Yaskawa INFORM job: SKRZYNIA_5040_180_STOPNI_10B_NEW.JBI

/JOB
//NAME SKRZYNIA_5040_180_STOPNI_10B_NEW
///FOLDERNAME 02-SKRZYNIE_JOBS
//POS
///NPOS 627,627,0,26,0,0
///TOOL 0
///POSTYPE PULSE
///PULSE
C00000=-21231,-51303,42314,2367,6591,-1439
C00001=-12854,-61498,-6635,149088,-29435,16513
C00002=84284,-61498,-6635,149088,14842,16513
C00003=84426,-61498,-62039,149088,14842,16513
C00004=84426,-61498,-83719,149088,14842,16513
C00005=40079,-25830,-61904,72398,37828,17494
C00006=40079,-25830,-61904,72398,37828,17494
C00007=38824,-23395,-60038,72349,38727,17731
C00008=41545,-22667,-59464,70826,37145,18191
C00009=40079,-25830,-61904,72398,37828,17494
C00010=40079,-23879,-31232,97616,36989,2612
C00011=40241,-22903,-30855,97033,36795,2952
C00012=39596,-21803,-29985,96678,37187,3182
C00013=41542,-21522,-29763,96797,35874,3054
C00014=40241,-22903,-30855,97033,36795,2952
C00015=44500,-22967,-34027,49689,40772,15208
C00016=44759,-21950,-33222,49364,40770,15399
C00017=43898,-20603,-32137,49608,41392,15289
C00018=45676,-20288,-31878,48567,40497,15854
C00019=44759,-21950,-33222,49364,40770,15399
C00020=50639,-31838,-53853,40430,42590,20636
C00021=47737,-42531,-47731,84740,46626,-3202
C00022=73324,-51450,-15857,136644,48513,-27329
C00023=28578,-31257,-33285,101874,54895,-3139
C00024=29101,-23166,-41439,93785,52323,3372
C00025=30342,-16402,-40775,90158,51109,6027
C00026=29555,-14242,-38855,90054,51607,6222
C00027=31304,-14182,-38798,89754,50458,6198
C00028=30342,-16402,-40775,90158,51109,6027
C00029=37840,-26567,-47806,97824,39338,5403
C00030=38314,-22656,-45541,96192,38787,6352
C00031=38740,-21749,-44817,95954,38481,6451
C00032=38106,-20505,-43805,95701,38856,6673
C00033=39920,-20274,-43616,95549,37666,6573
C00034=38740,-21749,-44817,95954,38481,6451
C00035=35154,-23288,-28184,89821,43405,2441
C00036=35403,-21021,-26397,89340,43215,2751
C00037=34678,-19569,-25213,89063,43699,2948
C00038=36545,-19419,-25091,89018,42427,2940
C00039=35403,-21021,-26397,89340,43215,2751
C00040=46673,-28267,-59493,36306,49500,22578
C00041=47298,-25083,-54483,36432,48421,22382
C00042=46134,-23276,-53085,36983,49197,22170
C00043=48093,-22778,-52692,35651,48513,22818
C00044=47298,-25083,-54483,36432,48421,22382
C00045=43000,-32780,-49011,53703,41088,15214
C00046=66148,-65994,-55487,105361,28212,-7739
C00047=66148,-65994,-55487,105361,28212,-7739
C00048=59848,-54778,-49507,133915,29212,-10807
C00049=45497,-38347,-41839,114412,32622,-465
C00050=46376,-32635,-46933,102993,29107,5780
C00051=46303,-28031,-46898,97061,28371,8976
C00052=45038,-26161,-45521,96183,29128,9541
C00053=46946,-25787,-45238,96120,27855,9431
C00054=46303,-28031,-46898,97061,28371,8976
C00055=45864,-17128,1685,129467,40696,-9274
C00056=46023,-15894,1830,128891,40053,-8896
C00057=45181,-14790,2774,128176,40341,-8535
C00058=46921,-14545,2986,129317,39465,-9073
C00059=45402,-17127,796,128656,40504,-8810
C00060=42828,-21985,-11573,106778,34538,-1929
C00061=43349,-21404,-11124,106831,34165,-1930
C00062=42250,-19876,-9917,105946,34757,-1485
C00063=44494,-19460,-9583,106781,33302,-1837
C00064=42797,-21858,-11474,106726,34550,-1903
C00065=42956,-14057,7354,88292,32197,-569
C00066=43438,-13569,7781,88275,31880,-510
C00067=42549,-12302,8904,87823,32462,-349
C00068=44721,-11883,9282,88161,31033,-316
C00069=42944,-14884,6642,88491,32210,-682
C00070=72417,-64226,-72669,53660,37323,27470
C00071=81480,-74508,-67932,111005,17511,3722
C00072=42492,-36415,-29790,92406,42740,11684
C00073=29699,-14901,-14062,86637,51249,15251
C00074=28921,-12904,-12269,86425,51786,15406
C00075=30978,-12767,-12144,86426,50380,15429
C00076=29506,-17416,-16239,86937,51377,15018
C00077=88410,-69609,-60867,139529,19008,-8209
C00078=62412,-62489,-12046,-12266,17816,34850
C00079=0,-52280,40443,0,6876,0
C00080=-681,-52632,38645,-5695,5489,-631
C00081=-17840,-61498,-6635,-149088,-29435,-16513
C00082=-84284,-61498,-6635,-149088,14842,-16513
C00083=-84426,-61498,-62039,-149088,14842,-16513
C00084=-84426,-61498,-83719,-149088,14842,-16513
C00085=-83351,-27062,-60322,-167360,37385,6517
C00086=-83351,-27062,-60322,-167360,37385,23281
C00087=-45097,-23850,-79932,-76262,26943,-22849
C00088=-48253,-15729,-73342,-71138,25693,-24842
C00089=-50302,-13076,-73239,-65836,25323,-27140
C00090=-49401,-11675,-71961,-66260,25816,-27133
C00091=-50608,-11574,-71867,-65226,25249,-27391
C00092=-49660,-13361,-73494,-66442,25615,-26975
C00093=-48242,-21102,-77802,-73044,25430,-23851
C00094=-42432,-29691,-46140,-101591,34194,-3953
C00095=-40467,-32259,-45349,-89481,35752,-6083
C00096=-35590,-22323,-38089,-87474,43148,-7978
C00097=-34853,-20780,-36847,-87247,43643,-8181
C00098=-37029,-20471,-36594,-86926,42180,-8224
C00099=-35503,-23333,-38886,-87700,43207,-7835
C00100=-41659,-25848,-37197,-61468,39541,-12344
C00101=-42019,-23363,-32043,-63110,38591,-11327
C00102=-41283,-22167,-31102,-63128,39154,-11341
C00103=-43189,-21868,-30866,-62281,38009,-11788
C00104=-40846,-25460,-35158,-62968,39555,-11455
C00105=-39561,-32409,-42051,-71473,38885,-9254
C00106=-88477,-67032,-53890,-125185,13082,17955
C00107=-90715,-66667,-50935,-152816,24533,28486
C00108=-30735,-26920,-32844,-95116,50209,-1071
C00109=-37180,-24683,-31930,-114741,47007,2943
C00110=-36407,-19634,-34656,-109847,45004,-453
C00111=-38352,-16604,-33863,-108521,43129,-1176
C00112=-37479,-14809,-32279,-108169,43576,-1482
C00113=-39395,-14487,-31992,-108361,42368,-1194
C00114=-37253,-18321,-35339,-108644,43916,-1187
C00115=-30948,-19486,-27368,-89515,49970,-2899
C00116=-32453,-17458,-25663,-89179,48933,-3088
C00117=-31896,-16151,-24534,-89028,49305,-3221
C00118=-33527,-16125,-24510,-88960,48196,-3202
C00119=-31291,-18911,-26892,-89421,49733,-2955
C00120=-32789,-14788,-10714,-75998,48642,-1904
C00121=-33953,-13481,-9550,-75758,47902,-2112
C00122=-33380,-12226,-8408,-75670,48319,-2157
C00123=-35020,-12164,-8351,-75529,47228,-2306
C00124=-33300,-14767,-10697,-75957,48300,-1949
C00125=-33300,-14767,-10697,-75957,48300,-1949
C00126=-33901,-13199,-7224,-76945,47663,-1266
C00127=-33178,-11617,-5779,-76815,48184,-1329
C00128=-35129,-11426,-5603,-76688,46886,-1497
C00129=-32900,-14718,-9841,-76444,48459,-1584
C00130=-46324,-38325,-53351,-48650,39022,-16558
C00131=-84678,-53272,-42524,-56273,5220,-14251
C00132=-79949,-57830,-54545,-43165,18800,-25262
C00133=-85199,-63426,-59279,-35356,8253,-25340
C00134=-43240,-40066,-69296,-76804,34492,-13950
C00135=-32352,-24302,-62495,-76398,48702,-17646
C00136=-33867,-19497,-59989,-74208,48202,-18898
C00137=-33043,-17469,-58279,-74274,48770,-19034
C00138=-35172,-17180,-58031,-73305,47532,-19251
C00139=-33150,-20833,-61090,-74721,48572,-18687
C00140=-32525,-19963,-22291,-97454,48417,-2656
C00141=-34479,-17146,-19937,-97221,47013,-2812
C00142=-33716,-15515,-18525,-96928,47480,-3025
C00143=-35357,-15455,-18472,-97073,46375,-2908
C00144=-33341,-18474,-21063,-97306,47817,-2759
C00145=-32838,-10388,7981,-94473,48357,2926
C00146=-33747,-9461,8037,-94117,47673,2571
C00147=-33094,-8062,9377,-93861,48090,2458
C00148=-34952,-7927,9507,-94260,46861,2543
C00149=-33010,-10379,7174,-94037,48174,2591
C00150=-36099,-20774,-22249,-70758,44565,-7624
C00151=-37926,-16067,-12890,-73276,42575,-5996
C00152=-37323,-14944,-11908,-73188,43017,-6038
C00153=-39053,-14785,-11769,-72915,41882,-6255
C00154=-37847,-19214,-17221,-72670,42783,-6386
C00155=-73757,-59015,-49060,-81128,32509,-3444
C00156=-66351,-49775,-22313,-121187,42752,19491
C00157=-38126,-18978,-6321,-103556,42156,4232
C00158=-39485,-17529,-8330,-90200,39091,223
C00159=-38315,-15563,-6658,-89669,39866,-39
C00160=-40130,-15376,-6497,-89855,38637,-21
C00161=-40610,-23081,-12745,-91737,38407,1092
C00162=-82794,-45547,-18103,-153793,26453,27163
C00163=-46099,-67236,-11725,-98004,28606,19827
C00164=275,-40498,62911,330,272,-175
C00165=-21231,-51303,42314,2367,6591,-1439
C00166=-12854,-61498,-6635,149088,-29435,16513
C00167=84284,-61498,-6635,149088,14842,16513
C00168=84426,-61498,-62039,149088,14842,16513
C00169=84426,-61498,-83719,149088,14842,16513
C00170=40079,-25830,-61904,72398,37828,17494
C00171=43542,-21744,-53414,85694,32141,12908
C00172=43538,-20959,-59091,78847,32551,16732
C00173=40079,-23879,-31232,97616,36989,2612
C00174=41069,-22296,-36683,87871,35939,7163
C00175=41069,-20857,-27994,94343,36275,3375
C00176=40241,-22903,-30855,97033,36795,2952
C00177=44500,-22967,-34027,49689,40772,15208
C00178=37674,-14410,-29425,54908,51799,12689
C00179=37617,-13106,-20810,58248,49229,10178
C00180=44759,-21950,-33222,49364,40770,15399
C00181=50639,-31838,-53853,40430,42590,20636
C00182=47737,-42531,-47731,84740,46626,-3202
C00183=78713,-49095,-28754,133607,38203,-24422
C00184=28578,-31257,-33285,101874,54895,-3139
C00185=29101,-23166,-41439,93785,52323,3372
C00186=31163,-13872,-34138,92103,50752,4440
C00187=31163,-14064,-41434,88282,50498,7326
C00188=30342,-16402,-40775,90158,51109,6027
C00189=37840,-26567,-47806,97824,39338,5403
C00190=38314,-22656,-45541,96192,38787,6352
C00191=39658,-19881,-39017,99036,38353,4498
C00192=39658,-20227,-46296,93241,37598,7980
C00193=38740,-21749,-44817,95954,38481,6451
C00194=35154,-23288,-28184,89821,43405,2441
C00195=36302,-20456,-32356,81251,42995,6506
C00196=36302,-19046,-24537,85721,42698,3608
C00197=35403,-21021,-26397,89340,43215,2751
C00198=46673,-28267,-59493,36306,49500,22578
C00199=35383,-14910,-45807,52457,59655,19882
C00200=35383,-15025,-38926,54776,56903,17744
C00201=47298,-25083,-54483,36432,48421,22382
C00202=43000,-32780,-49011,53703,41088,15214
C00203=90538,-65158,-52413,145953,6697,-22013
C00204=90538,-65158,-52413,145953,6697,-22013
C00205=59848,-54778,-49507,133915,29212,-10807
C00206=45497,-38347,-41839,114412,32622,-465
C00207=46376,-32635,-46933,102993,29107,5780
C00208=38443,-20223,-37840,96971,39567,10287
C00209=38443,-20698,-44956,91660,38993,13539
C00210=46303,-28031,-46898,97061,28371,8976
C00211=45864,-17128,1685,129467,40696,-9274
C00212=38069,-7942,12691,120284,49952,-5070
C00213=38069,-11604,1369,116685,47266,-2469
C00214=45402,-17127,796,128656,40504,-8810
C00215=42828,-21985,-11573,106778,34538,-1929
C00216=33281,-15275,-13406,92642,47209,4970
C00217=33281,-12456,-2996,97026,47894,1870
C00218=42797,-21858,-11474,106726,34550,-1903
C00219=42956,-14057,7354,88292,32197,-569
C00220=35915,-8349,8335,81338,43542,2014
C00221=35915,-4149,20758,86814,43229,-1568
C00222=42944,-14884,6642,88491,32210,-682
C00223=72417,-64226,-72669,53660,37323,27470
C00224=81480,-74508,-67932,111005,17511,3722
C00225=31559,-23192,-27729,97069,50041,14774
C00226=34278,-17590,-29530,108925,47275,14558
C00227=34921,-13948,-26935,108215,46513,15013
C00228=34921,-14719,-34056,104413,45059,17611
C00229=33936,-16225,-25259,110400,48238,13526
C00230=30729,-14807,-22031,91030,50318,16982
C00231=30729,-13019,-13516,94566,50766,14318
C00232=88410,-69609,-60867,139529,19008,-8209
C00233=62412,-62489,-12046,-12266,17816,34850
C00234=0,-52280,40443,0,6876,0
C00235=-681,-52632,38645,-5695,5489,-631
C00236=-17840,-61498,-6635,-149088,-29435,-16513
C00237=-84284,-61498,-6635,-149088,14842,-16513
C00238=-84426,-61498,-62039,-149088,14842,-16513
C00239=-84426,-61498,-83719,-149088,14842,-16513
C00240=-83351,-27062,-60322,-167360,37385,6517
C00241=-83351,-27062,-60322,-167360,37385,23281
C00242=-45097,-23850,-79932,-76262,26943,-22849
C00243=-48253,-15729,-73342,-71138,25693,-24842
C00244=-42869,-6204,-67496,-75794,33821,-25861
C00245=-42869,-3205,-70686,-69723,34977,-29338
C00246=-49660,-13361,-73494,-66442,25615,-26975
C00247=-48242,-21102,-77802,-73044,25430,-23851
C00248=-42432,-29691,-46140,-101591,34194,-3953
C00249=-40467,-32259,-45349,-89481,35752,-6083
C00250=-32032,-15700,-34761,-86363,49905,-9645
C00251=-32032,-14866,-27372,-89947,49973,-6979
C00252=-35503,-23333,-38886,-87700,43207,-7835
C00253=-41659,-25848,-37197,-61468,39541,-12344
C00254=-32550,-13183,-23016,-68651,53358,-8526
C00255=-34023,-12481,-22084,-63241,53452,-9524
C00256=-40846,-25460,-35158,-62968,39555,-11455
C00257=-39561,-32409,-42051,-71473,38885,-9254
C00258=-88477,-67032,-53890,-125185,13082,17955
C00259=-90715,-66667,-50935,-152816,24533,28486
C00260=-30735,-26920,-32844,-95116,50209,-1071
C00261=-37180,-24683,-31930,-114741,47007,2943
C00262=-36407,-19634,-34656,-109847,45004,-453
C00263=-39264,-14095,-28560,-110319,43249,69
C00264=-39254,-14742,-35710,-105973,41627,-2729
C00265=-37253,-18321,-35339,-108644,43916,-1187
C00266=-30948,-19486,-27368,-89515,49970,-2899
C00267=-33188,-17217,-33290,-80523,49125,-7157
C00268=-33231,-16133,-25752,-84153,48705,-4513
C00269=-31291,-18911,-26892,-89421,49733,-2955
C00270=-32789,-14788,-10714,-75998,48642,-1904
C00271=-32456,-10000,-8763,-74569,51725,-2878
C00272=-32456,-7502,814,-78111,50801,-165
C00273=-33300,-14767,-10697,-75957,48300,-1949
C00274=-33300,-14767,-10697,-75957,48300,-1949
C00275=-31039,-7597,-4415,-75714,54029,-1891
C00276=-31745,-5891,1281,-74609,53027,-1007
C00277=-32900,-14718,-9841,-76444,48459,-1584
C00278=-46324,-38325,-53351,-48650,39022,-16558
C00279=-84678,-53272,-42524,-56273,5220,-14251
C00280=-79949,-57830,-54545,-43165,18800,-25262
C00281=-85199,-63426,-59279,-35356,8253,-25340
C00282=-43240,-40066,-69296,-76804,34492,-13950
C00283=-32352,-24302,-62495,-76398,48702,-17646
C00284=-34311,-15084,-43386,-89458,46770,-12174
C00285=-34303,-14562,-49859,-85086,46777,-15220
C00286=-33150,-20833,-61090,-74721,48572,-18687
C00287=-32525,-19963,-22291,-97454,48417,-2656
C00288=-35706,-13608,-12356,-102024,46946,-662
C00289=-35706,-15621,-21438,-97808,45877,-3577
C00290=-33341,-18474,-21063,-97306,47817,-2759
C00291=-32838,-10388,7981,-94473,48357,2926
C00292=-33093,-7396,5806,-90907,49596,566
C00293=-33114,-3922,16616,-94789,50065,3444
C00294=-33010,-10379,7174,-94037,48174,2591
C00295=-36099,-20774,-22249,-70758,44565,-7624
C00296=-34715,-11750,-12273,-72011,49148,-6727
C00297=-34715,-9605,-3694,-75523,48112,-4187
C00298=-37847,-19214,-17221,-72670,42783,-6386
C00299=-73757,-59015,-49060,-81128,30370,-3444
C00300=-66351,-49775,-22313,-115582,40632,19491
C00301=-39230,-13378,9505,-118180,46878,7841
C00302=-45382,-7236,12023,-133378,48537,9962
C00303=-45404,-10871,608,-130166,44845,7725
C00304=-39289,-13633,5656,-114159,44810,6160
C00305=-38323,-13232,3563,-106275,42852,3854
C00306=-39624,-12309,2722,-105485,41613,3229
C00307=-39624,-8328,14658,-110578,43519,6514
C00308=-36264,-16485,7382,-110054,45980,6615
C00309=-44249,-32643,-4456,-118298,43922,12613
C00310=-31781,-48654,10305,-108801,40875,18482
C00311=275,-40498,62911,330,272,-175
C00312=-21231,-51303,42314,2367,6591,-1439
C00313=-12854,-61498,-6635,149088,-29435,16513
C00314=32880,-72586,-50560,79734,53940,25582
C00315=76664,-93599,-96338,114349,24908,7990
C00316=72545,-76403,-90681,98079,12187,16258
C00317=68435,-42241,-79282,43384,21203,43145
C00318=65057,-16377,-54230,51764,24572,24912
C00319=65057,-16377,-54230,51764,24572,24912
C00320=63338,-14509,-52578,53100,25585,24479
C00321=65493,-13068,-51269,50530,24633,25485
C00322=65057,-16377,-54230,51764,24572,24912
C00323=65057,-15356,-24189,99795,20011,765
C00324=64877,-14372,-23690,98704,20045,1316
C00325=64002,-13489,-22890,98156,20604,1621
C00326=65592,-12702,-22173,98357,19527,1466
C00327=64877,-14372,-23690,98704,20045,1316
C00328=68341,-13254,-25781,29903,31229,25524
C00329=68283,-12212,-24821,29865,31356,25548
C00330=67188,-11145,-23825,30867,31841,25051
C00331=68624,-10377,-23095,29361,31405,25809
C00332=68283,-12212,-24821,29865,31356,25548
C00333=67373,-28813,-51747,26561,36937,27500
C00334=65665,-56911,-59086,75825,31170,1181
C00335=86238,-56758,-47218,93606,16664,-7096
C00336=86238,-56758,-47218,93606,16664,-7096
C00337=58162,-25487,-29222,106212,35121,-6052
C00338=54729,-17550,-36821,90686,35172,3055
C00339=53879,-10723,-35593,84994,35691,6442
C00340=52628,-8898,-33837,85063,36512,6546
C00341=54193,-8333,-33282,84633,35489,6620
C00342=53879,-10723,-35593,84994,35691,6442
C00343=63265,-18185,-41125,95483,22448,4389
C00344=62561,-14368,-38517,92984,22773,5727
C00345=62689,-13396,-37636,92694,22678,5861
C00346=61812,-12400,-36718,92465,23238,6064
C00347=63331,-11679,-36046,92201,22238,6052
C00348=62689,-13396,-37636,92694,22678,5861
C00349=60836,-16142,-22303,87853,25853,3109
C00350=60346,-13901,-20318,87240,26185,3441
C00351=59279,-12702,-19226,86999,26911,3593
C00352=60868,-12050,-18626,86765,25831,3679
C00353=60346,-13901,-20318,87240,26185,3441
C00354=71174,-16943,-50501,16787,44328,31924
C00355=70846,-13961,-45205,17496,43056,31510
C00356=69412,-12602,-43961,18675,43507,30969
C00357=70949,-11616,-43043,17320,43301,31610
C00358=70846,-13961,-45205,17496,43056,31510
C00359=66765,-25643,-43957,33958,30926,25005
C00360=89904,-51519,-74342,14421,36812,44678
C00361=59533,-60921,-66479,83565,41795,11392
C00362=74572,-27669,-34920,136415,14797,-11887
C00363=72479,-21736,-38943,108586,11547,1590
C00364=70901,-17325,-38411,94105,11830,8638
C00365=69318,-15905,-37172,92885,12849,9347
C00366=70820,-15051,-36412,92531,11846,9399
C00367=70901,-17325,-38411,94105,11830,8638
C00368=70927,-7523,10343,151197,29871,-19432
C00369=70517,-6236,10737,150221,29352,-18933
C00370=69462,-5331,11645,148944,29606,-18324
C00371=70849,-4645,12343,150548,29173,-19084
C00372=70402,-7634,9356,150158,29478,-18907
C00373=68660,-13051,-4106,122816,18275,-8999
C00374=68895,-12351,-3471,122899,18094,-9031
C00375=67458,-11121,-2337,120787,18802,-8043
C00376=69212,-10147,-1425,122703,17774,-8922
C00377=68590,-12934,-4000,122687,18305,-8939
C00378=67960,-5141,15741,92957,15720,-628
C00379=68207,-4523,16370,92944,15555,-601
C00380=67051,-3465,17460,92338,16311,-404
C00381=68762,-2475,18496,92897,15183,-531
C00382=68227,-5981,14898,93242,15553,-745
C00383=75423,-38775,-29488,68062,11357,11878
C00384=83800,-53438,-37305,103753,25026,-1265
C00385=73693,-43023,-29306,101200,31062,8332
C00386=57182,-8361,13896,122065,42938,1264
C00387=54175,-4244,10116,111777,38351,4895
C00388=53015,-2664,11762,111180,39035,5172
C00389=54334,-2350,12093,111780,38228,4906
C00390=54175,-4244,10116,111777,38351,4895
C00391=89016,-59505,-36896,143842,20811,-11822
C00392=0,-52280,40443,0,6876,0
C00393=-681,-52632,38645,-5695,5489,-631
C00394=-17840,-61498,-6635,-149088,-29435,-16513
C00395=-84284,-61498,-6635,-149088,14842,-16513
C00396=-57949,-92832,-68327,-119114,39180,-13331
C00397=-51160,-78996,-68705,-103851,38676,-21739
C00398=-70129,-12201,-70194,-45988,15849,-32683
C00399=-70861,-4247,-62448,-43170,16032,-33903
C00400=-72229,-1292,-61598,-37253,16795,-36501
C00401=-71164,-286,-60510,-39045,17142,-35862
C00402=-72168,114,-60071,-37345,16819,-36474
C00403=-71747,-1710,-62044,-38091,16943,-36199
C00404=-72086,-8949,-67137,-41785,15362,-34318
C00405=-68226,-19972,-38714,-103620,16923,-1218
C00406=-67549,-22986,-38612,-80975,17520,-9124
C00407=-60286,-14955,-31870,-81576,26630,-9634
C00408=-59206,-13694,-30736,-81541,27366,-9725
C00409=-61026,-12796,-29913,-80837,26167,-9971
C00410=-60502,-15936,-32740,-81790,26471,-9505
C00411=-66711,-16726,-29834,-42060,26790,-21996
C00412=-66477,-14329,-24475,-44917,25565,-20507
C00413=-65503,-13376,-23611,-45716,26132,-20127
C00414=-67048,-12587,-22889,-44009,25442,-20959
C00415=-66009,-16611,-27996,-44380,26285,-20808
C00416=-67084,-23473,-35621,-52822,22843,-18344
C00417=-54372,-63877,-56403,-90862,27079,1323
C00418=-55608,-75012,-34654,-126966,55573,20814
C00419=-55608,-75012,-34654,-126966,55573,20814
C00420=-58069,-20780,-28125,-95622,31565,-134
C00421=-62818,-16895,-25617,-123146,31403,8811
C00422=-60301,-12189,-28106,-114654,29999,4030
C00423=-61167,-8731,-26593,-112607,28768,2985
C00424=-59960,-7252,-25135,-111997,29446,2563
C00425=-61574,-6413,-24296,-112502,28453,2957
C00426=-60636,-10677,-28466,-112685,29164,2987
C00427=-55814,-13636,-22293,-87541,33030,-3263
C00428=-56566,-11270,-20110,-87077,32519,-3496
C00429=-55709,-10167,-19066,-86969,33101,-3589
C00430=-57154,-9687,-18605,-86794,32120,-3632
C00431=-55949,-12989,-21706,-87412,32939,-3330
C00432=-57109,-8613,-4995,-71756,32687,-5152
C00433=-57764,-7017,-3429,-71410,32292,-5358
C00434=-56909,-5946,-2356,-71529,32873,-5273
C00435=-58347,-5433,-1836,-71115,31941,-5534
C00436=-57555,-8453,-4841,-71622,32398,-5235
C00437=-57555,-8453,-4841,-71622,32398,-5235
C00438=-57844,-6749,-1100,-73475,31868,-4209
C00439=-56760,-5394,262,-73573,32605,-4123
C00440=-58439,-4668,1002,-73167,31507,-4396
C00441=-57269,-8513,-4090,-72514,32435,-4729
C00442=-74194,-26905,-45748,-21164,30431,-30370
C00443=-93036,-61583,-83098,-4972,39040,-38907
C00444=-93036,-61583,-83098,-4972,39040,-38907
C00445=-71878,-28414,-61729,-48672,19032,-25171
C00446=-58025,-17185,-56692,-61796,34178,-22014
C00447=-58138,-12270,-53641,-59720,34855,-23185
C00448=-56898,-10637,-52111,-60384,35596,-23031
C00449=-58712,-9745,-51261,-58987,34681,-23500
C00450=-57851,-13714,-54968,-60141,34926,-22995
C00451=-57767,-13689,-16896,-100181,31334,-836
C00452=-58645,-10437,-13885,-99794,30663,-1040
C00453=-57513,-9065,-12573,-99347,31388,-1300
C00454=-58947,-8556,-12078,-99591,30423,-1148
C00455=-58031,-12031,-15383,-99926,31110,-974
C00456=-57646,-4162,14084,-101426,32077,4804
C00457=-58050,-2999,14481,-100683,31666,4357
C00458=-57067,-1784,15765,-100255,32298,4198
C00459=-58672,-1130,16464,-100866,31256,4407
C00460=-57676,-4116,13320,-100600,31921,4338
C00461=-61201,-13510,-16039,-60848,29053,-13371
C00462=-61885,-8475,-5914,-65722,27292,-10768
C00463=-61040,-7537,-4993,-65975,27855,-10622
C00464=-62506,-6917,-4380,-65230,26947,-11038
C00465=-62587,-11561,-10517,-63923,27184,-11731
C00466=-69972,-70945,-58827,-87515,35615,-17
C00467=-69972,-70945,-58827,-87515,35615,-17
C00468=-64053,-11295,342,-114563,25508,8776
C00469=-64305,-9514,-1154,-92513,22236,350
C00470=-62690,-7882,422,-91839,23314,70
C00471=-64201,-7220,1072,-92034,22288,112
C00472=-67149,-14673,-5883,-94845,20391,1413
C00473=-66017,-67071,-29713,-134523,32873,22112
C00474=-46099,-67236,-11725,-98004,28606,19827
C00475=275,-40498,62911,330,272,-175
C00476=-21231,-51303,42314,2367,6591,-1439
C00477=-12854,-61498,-6635,149088,-29435,16513
C00478=84284,-61498,-6635,149088,14842,16513
C00479=84426,-61498,-62039,149088,14842,16513
C00480=84426,-61498,-83719,149088,14842,16513
C00481=65057,-16377,-54230,51764,24572,24912
C00482=84197,-12836,-45810,-45141,8815,68584
C00483=84197,-12041,-51210,-30828,12194,61758
C00484=65057,-15356,-24189,99795,20011,765
C00485=74080,-15423,-30907,69143,7686,14038
C00486=74080,-14352,-23480,100923,7503,-991
C00487=64877,-14372,-23690,98704,20045,1316
C00488=68341,-13254,-25781,29903,31229,25524
C00489=74439,-11496,-26749,13621,29642,33649
C00490=74439,-10401,-19085,15788,25340,32499
C00491=68283,-12212,-24821,29865,31356,25548
C00492=75452,-19560,-44582,17787,36745,31835
C00493=68183,-44834,-62310,40554,34116,19994
C00494=94103,-63119,-69903,16230,17694,31762
C00495=91219,-55958,-51219,93435,14423,-1742
C00496=58162,-25487,-29222,106212,35121,-6052
C00497=54729,-17550,-36821,90686,35172,3055
C00498=70769,-15160,-35297,83470,11760,4000
C00499=70769,-15377,-40609,67973,12489,11436
C00500=53879,-10723,-35593,84994,35691,6442
C00501=63265,-18185,-41125,95483,22448,4389
C00502=62561,-14368,-38517,92984,22773,5727
C00503=77715,-13962,-33882,144680,4496,-21400
C00504=77806,-14046,-41277,60589,2532,18064
C00505=62689,-13396,-37636,92694,22678,5861
C00506=60836,-16142,-22303,87853,25853,3109
C00507=74678,-16514,-29029,42946,9451,23276
C00508=74678,-15315,-21920,65026,7151,12815
C00509=60346,-13901,-20318,87240,26185,3441
C00510=71174,-16943,-50501,16787,44328,31924
C00511=80494,-13102,-44599,-1731,38384,44653
C00512=80494,-13295,-38861,-1907,34285,44756
C00513=70846,-13961,-45205,17496,43056,31510
C00514=69645,-22678,-41665,30358,30421,26767
C00515=81017,-78801,-66317,80675,7786,2447
C00516=81017,-78801,-66317,80675,7786,2447
C00517=74572,-27669,-34920,136415,14797,-11887
C00518=72479,-21736,-38943,108586,11547,1590
C00519=76162,-15538,-34076,119407,5153,-4143
C00520=76225,-15803,-40874,66675,4586,20654
C00521=70901,-17325,-38411,94105,11830,8638
C00522=70927,-7523,10343,151197,29871,-19432
C00523=75273,-951,23395,164730,33684,-27271
C00524=75257,-4812,11918,163197,28775,-26429
C00525=70402,-7634,9356,150158,29478,-18907
C00526=68660,-13051,-4106,122816,18275,-8999
C00527=75422,-13779,-12311,124767,7049,-10125
C00528=75402,-11409,-3274,143452,10422,-18986
C00529=68590,-12934,-4000,122687,18305,-8939
C00530=67960,-5141,15741,92957,15720,-628
C00531=77005,-5383,11265,73049,3770,10304
C00532=77005,-1367,23224,135174,5603,-18901
C00533=68227,-5981,14898,93242,15553,-745
C00534=83595,-66668,-34414,154325,14846,-28455
C00535=83596,-66666,-34415,154326,14845,-28454
C00536=69137,-30288,-25983,94330,24536,11676
C00537=63448,-5639,10903,136482,36601,-23409
C00538=72869,1541,21011,161481,40400,-32944
C00539=75019,3768,21884,166311,43242,-33805
C00540=75946,3919,31956,167866,49928,-34763
C00541=66712,-14281,-1549,117281,20128,-19574
C00542=71147,-20912,-26201,58115,12192,12177
C00543=72038,-15960,-22039,53337,12147,14456
C00544=72038,-13517,-11162,79650,10019,1887
C00545=70769,-47931,-32777,112213,25945,2479
C00546=17178,-50520,12136,39169,20391,2344
C00547=-681,-52632,38645,-5695,5489,-631
C00548=-17840,-61498,-6635,-149088,-29435,-16513
C00549=-84284,-61498,-6635,-149088,14842,-16513
C00550=-84426,-61498,-62039,-149088,14842,-16513
C00551=-84426,-61498,-83719,-149088,14842,-16513
C00552=-83351,-27062,-60322,-167360,37385,6517
C00553=-83351,-27062,-60322,-167360,37385,23281
C00554=-70129,-12201,-70194,-45988,15849,-32683
C00555=-70861,-4247,-62448,-43170,16032,-33903
C00556=-76882,43,-60950,-14294,14755,-45201
C00557=-76882,3984,-64926,-10429,20329,-47102
C00558=-71747,-1710,-62044,-38091,16943,-36199
C00559=-72086,-8949,-67137,-41785,15362,-34318
C00560=-68226,-19972,-38714,-103620,16923,-1218
C00561=-67549,-22986,-38612,-80975,17520,-9124
C00562=-69143,-15166,-34287,-68804,15212,-14794
C00563=-69143,-14592,-28782,-80821,14459,-8960
C00564=-60502,-15936,-32740,-81790,26471,-9505
C00565=-66711,-16726,-29834,-42060,26790,-21996
C00566=-75652,-13136,-22972,-17539,18443,-33643
C00567=-76393,-11602,-18975,-13556,19574,-34543
C00568=-66009,-16611,-27996,-44380,26285,-20808
C00569=-61601,-28306,-39228,-59626,25389,-15050
C00570=-72315,-63222,-70224,-69600,33305,-10426
C00571=-72315,-63222,-70224,-69600,33305,-10426
C00572=-58069,-20780,-28125,-95622,31565,-134
C00573=-62818,-16895,-25617,-123146,31403,8811
C00574=-60301,-12189,-28106,-114654,29999,4030
C00575=-75089,-9933,-24682,-148597,14783,22922
C00576=-75089,-10642,-34451,-132584,9653,15243
C00577=-60636,-10677,-28466,-112685,29164,2987
C00578=-55814,-13636,-22293,-87541,33030,-3263
C00579=-73301,-16058,-32281,-44459,12702,-22095
C00580=-73339,-15052,-25249,-60236,10249,-14543
C00581=-55949,-12989,-21706,-87412,32939,-3330
C00582=-57109,-8613,-4995,-71756,32687,-5152
C00583=-71674,-10355,-9102,-48278,15013,-17468
C00584=-71670,-8088,-356,-62615,12652,-10541
C00585=-57555,-8453,-4841,-71622,32398,-5235
C00586=-57555,-8453,-4841,-71622,32398,-5235
C00587=-73349,-10209,-7254,-46090,12597,-18565
C00588=-73349,-7867,1452,-63091,10217,-10432
C00589=-57269,-8513,-4090,-72514,32435,-4729
C00590=-74194,-26905,-45748,-21164,30431,-30370
C00591=-76007,-77202,-67157,-59280,11041,-11579
C00592=-76006,-77203,-67157,-59281,11043,-11581
C00593=-53398,-42726,-55849,-45492,34374,-18069
C00594=-71878,-28414,-61729,-48672,19032,-25171
C00595=-58025,-17185,-56692,-61796,34178,-22014
C00596=-77553,-14661,-43008,-35465,5780,-31120
C00597=-77553,-14004,-50514,-17997,10868,-39389
C00598=-57851,-13714,-54968,-60141,34926,-22995
C00599=-57767,-13689,-16896,-100181,31334,-836
C00600=-74769,-11126,-10073,-142523,13426,19686
C00601=-74753,-12848,-17783,-130765,10301,14051
C00602=-58031,-12031,-15383,-99926,31110,-974
C00603=-57646,-4162,14084,-101426,32077,4804
C00604=-72179,-7124,6017,-115427,12582,9833
C00605=-72179,-4103,15503,-129018,15105,16401
C00606=-57676,-4116,13320,-100600,31921,4338
C00607=-61201,-13510,-16039,-60848,29053,-13371
C00608=-74136,-10643,-11909,-32993,14820,-27251
C00609=-74162,-8377,-2780,-45377,11297,-21290
C00610=-62587,-11561,-10517,-63923,27184,-11731
C00611=-68334,-63389,-52515,-83837,33201,-1739
C00612=-68334,-63389,-52515,-83837,33201,-1739
C00613=-64053,-11295,342,-114563,25508,8776
C00614=-76017,6008,33610,-165984,45639,36413
C00615=-74239,7065,32887,-163372,44700,35065
C00616=-74142,3045,20239,-161993,39159,34198
C00617=-75119,4045,29308,-164063,44402,35406
C00618=-79833,-9558,5437,-165750,9898,43323
C00619=-74932,-11787,84,-126218,10763,24539
C00620=-75231,-7555,5870,-137998,10766,30530
C00621=-75231,-3987,16941,-149127,14978,35883
C00622=-77761,-13214,8113,-156332,15145,39163
C00623=-65551,-48104,-28924,-114827,24376,11665
C00624=-51220,-46814,3045,-130057,64886,23876
C00625=-46099,-67236,-11725,-98004,28606,19827
C00626=275,-40498,62911,330,272,-175
BC00000=467225
BC00001=513669
BC00002=494109
BC00003=467540
BC00004=467540
BC00005=478876
BC00006=478876
BC00007=478876
BC00008=478876
BC00009=478876
BC00010=478876
BC00011=478876
BC00012=478876
BC00013=478876
BC00014=478876
BC00015=478876
BC00016=478876
BC00017=478876
BC00018=478876
BC00019=478876
BC00020=478876
BC00021=481980
BC00022=563952
BC00023=606256
BC00024=606256
BC00025=606252
BC00026=606252
BC00027=606252
BC00028=606252
BC00029=654662
BC00030=654618
BC00031=654618
BC00032=654618
BC00033=654618
BC00034=654618
BC00035=654618
BC00036=654618
BC00037=654618
BC00038=654618
BC00039=654618
BC00040=686402
BC00041=686402
BC00042=686350
BC00043=686350
BC00044=686402
BC00045=652574
BC00046=648164
BC00047=761837
BC00048=784046
BC00049=784046
BC00050=784046
BC00051=784046
BC00052=784046
BC00053=784046
BC00054=784046
BC00055=784046
BC00056=784046
BC00057=784046
BC00058=784046
BC00059=784046
BC00060=821134
BC00061=821134
BC00062=821134
BC00063=821134
BC00064=821134
BC00065=821134
BC00066=821134
BC00067=821134
BC00068=821134
BC00069=821134
BC00070=849627
BC00071=991666
BC00072=955683
BC00073=955683
BC00074=955683
BC00075=955683
BC00076=955683
BC00077=991666
BC00078=856383
BC00079=828403
BC00080=518986
BC00081=509920
BC00082=467540
BC00083=467540
BC00084=467540
BC00085=521167
BC00086=520352
BC00087=535759
BC00088=535759
BC00089=535757
BC00090=535757
BC00091=535757
BC00092=535757
BC00093=535757
BC00094=485653
BC00095=485653
BC00096=485653
BC00097=485653
BC00098=485653
BC00099=485653
BC00100=485653
BC00101=485653
BC00102=485653
BC00103=485653
BC00104=485653
BC00105=485653
BC00106=485653
BC00107=615112
BC00108=615112
BC00109=615112
BC00110=615112
BC00111=615112
BC00112=615112
BC00113=615112
BC00114=615112
BC00115=615112
BC00116=615112
BC00117=615112
BC00118=615112
BC00119=615112
BC00120=615112
BC00121=615112
BC00122=615112
BC00123=615112
BC00124=615112
BC00125=658076
BC00126=658076
BC00127=658076
BC00128=658076
BC00129=658076
BC00130=655680
BC00131=643721
BC00132=643721
BC00133=793396
BC00134=799070
BC00135=799070
BC00136=799070
BC00137=799070
BC00138=799070
BC00139=799070
BC00140=799070
BC00141=799070
BC00142=799070
BC00143=799070
BC00144=799070
BC00145=799070
BC00146=799070
BC00147=799070
BC00148=799070
BC00149=799070
BC00150=845667
BC00151=845667
BC00152=845667
BC00153=845667
BC00154=845667
BC00155=845667
BC00156=945519
BC00157=945519
BC00158=945519
BC00159=945519
BC00160=945519
BC00161=945519
BC00162=945519
BC00163=895479
BC00164=639407
BC00165=467225
BC00166=513669
BC00167=494109
BC00168=467540
BC00169=467540
BC00170=478876
BC00171=478876
BC00172=478876
BC00173=478876
BC00174=478876
BC00175=478876
BC00176=478876
BC00177=478876
BC00178=478876
BC00179=478876
BC00180=478876
BC00181=478876
BC00182=481980
BC00183=578133
BC00184=606256
BC00185=606256
BC00186=606252
BC00187=606252
BC00188=606252
BC00189=654662
BC00190=654618
BC00191=654618
BC00192=654618
BC00193=654618
BC00194=654618
BC00195=654618
BC00196=654618
BC00197=654618
BC00198=686402
BC00199=686402
BC00200=686402
BC00201=686402
BC00202=652574
BC00203=641414
BC00204=715810
BC00205=784046
BC00206=784046
BC00207=784046
BC00208=784046
BC00209=784046
BC00210=784046
BC00211=784046
BC00212=784043
BC00213=784043
BC00214=784046
BC00215=821134
BC00216=821134
BC00217=821134
BC00218=821134
BC00219=821134
BC00220=821134
BC00221=821134
BC00222=821134
BC00223=849627
BC00224=990121
BC00225=990121
BC00226=990121
BC00227=990121
BC00228=990121
BC00229=990121
BC00230=974760
BC00231=974760
BC00232=979650
BC00233=855778
BC00234=786675
BC00235=518986
BC00236=509920
BC00237=467540
BC00238=467540
BC00239=467540
BC00240=521167
BC00241=520352
BC00242=535759
BC00243=535759
BC00244=535757
BC00245=535757
BC00246=535757
BC00247=535757
BC00248=485653
BC00249=485653
BC00250=485653
BC00251=485653
BC00252=485653
BC00253=485653
BC00254=485653
BC00255=485653
BC00256=485653
BC00257=485653
BC00258=485653
BC00259=615112
BC00260=615112
BC00261=615112
BC00262=615112
BC00263=615112
BC00264=615112
BC00265=615112
BC00266=615112
BC00267=615112
BC00268=615112
BC00269=615112
BC00270=615112
BC00271=615112
BC00272=615112
BC00273=615112
BC00274=658076
BC00275=658076
BC00276=658076
BC00277=658076
BC00278=655680
BC00279=643721
BC00280=643721
BC00281=793396
BC00282=799070
BC00283=799070
BC00284=799070
BC00285=799070
BC00286=799070
BC00287=799070
BC00288=799070
BC00289=799070
BC00290=799070
BC00291=799070
BC00292=799070
BC00293=799070
BC00294=799070
BC00295=845667
BC00296=845667
BC00297=845667
BC00298=845667
BC00299=845667
BC00300=944991
BC00301=940590
BC00302=940590
BC00303=940590
BC00304=940590
BC00305=949966
BC00306=949966
BC00307=949966
BC00308=949966
BC00309=938866
BC00310=879370
BC00311=639407
BC00312=467225
BC00313=513669
BC00314=542621
BC00315=535309
BC00316=478364
BC00317=478364
BC00318=478876
BC00319=478876
BC00320=478876
BC00321=478876
BC00322=478876
BC00323=478876
BC00324=478876
BC00325=478876
BC00326=478876
BC00327=478876
BC00328=478876
BC00329=478876
BC00330=478876
BC00331=478876
BC00332=478876
BC00333=478876
BC00334=480759
BC00335=480759
BC00336=560395
BC00337=606256
BC00338=606256
BC00339=606252
BC00340=606252
BC00341=606252
BC00342=606252
BC00343=654662
BC00344=654618
BC00345=654618
BC00346=654618
BC00347=654618
BC00348=654618
BC00349=654618
BC00350=654618
BC00351=654618
BC00352=654618
BC00353=654618
BC00354=686402
BC00355=686402
BC00356=686350
BC00357=686350
BC00358=686402
BC00359=652574
BC00360=652574
BC00361=774850
BC00362=784046
BC00363=784046
BC00364=784046
BC00365=784046
BC00366=784046
BC00367=784046
BC00368=784046
BC00369=784046
BC00370=784046
BC00371=784046
BC00372=784046
BC00373=821134
BC00374=821134
BC00375=821134
BC00376=821134
BC00377=821134
BC00378=821134
BC00379=821134
BC00380=821134
BC00381=821134
BC00382=821134
BC00383=821134
BC00384=846623
BC00385=955683
BC00386=955683
BC00387=955683
BC00388=955683
BC00389=955683
BC00390=955683
BC00391=955974
BC00392=795359
BC00393=518986
BC00394=509920
BC00395=467540
BC00396=497868
BC00397=497868
BC00398=535759
BC00399=535759
BC00400=535757
BC00401=535757
BC00402=535757
BC00403=535757
BC00404=535757
BC00405=485653
BC00406=485653
BC00407=485653
BC00408=485653
BC00409=485653
BC00410=485653
BC00411=485653
BC00412=485653
BC00413=485653
BC00414=485653
BC00415=485653
BC00416=485653
BC00417=485653
BC00418=485653
BC00419=601945
BC00420=615112
BC00421=615112
BC00422=615112
BC00423=615112
BC00424=615112
BC00425=615112
BC00426=615112
BC00427=615112
BC00428=615112
BC00429=615112
BC00430=615112
BC00431=615112
BC00432=615112
BC00433=615112
BC00434=615112
BC00435=615112
BC00436=615112
BC00437=658076
BC00438=658076
BC00439=658076
BC00440=658076
BC00441=658076
BC00442=655680
BC00443=655680
BC00444=765678
BC00445=799070
BC00446=799070
BC00447=799070
BC00448=799070
BC00449=799070
BC00450=799070
BC00451=799070
BC00452=799070
BC00453=799070
BC00454=799070
BC00455=799070
BC00456=799070
BC00457=799070
BC00458=799070
BC00459=799070
BC00460=799070
BC00461=845667
BC00462=845667
BC00463=845667
BC00464=845667
BC00465=845667
BC00466=845667
BC00467=977957
BC00468=945519
BC00469=945519
BC00470=945519
BC00471=945519
BC00472=945519
BC00473=930158
BC00474=895479
BC00475=639407
BC00476=467225
BC00477=513669
BC00478=494109
BC00479=467540
BC00480=467540
BC00481=478876
BC00482=478876
BC00483=478876
BC00484=478876
BC00485=478876
BC00486=478876
BC00487=478876
BC00488=478876
BC00489=478876
BC00490=478876
BC00491=478876
BC00492=478876
BC00493=479530
BC00494=502776
BC00495=571156
BC00496=606256
BC00497=606256
BC00498=606252
BC00499=606252
BC00500=606252
BC00501=654662
BC00502=654618
BC00503=654618
BC00504=654618
BC00505=654618
BC00506=654618
BC00507=654618
BC00508=654618
BC00509=654618
BC00510=686402
BC00511=686402
BC00512=686402
BC00513=686402
BC00514=652574
BC00515=654591
BC00516=763025
BC00517=784046
BC00518=784046
BC00519=784046
BC00520=784046
BC00521=784046
BC00522=784046
BC00523=784043
BC00524=784043
BC00525=784046
BC00526=821134
BC00527=821134
BC00528=821134
BC00529=821134
BC00530=821134
BC00531=821134
BC00532=821134
BC00533=821134
BC00534=821134
BC00535=928534
BC00536=952873
BC00537=943447
BC00538=948826
BC00539=948826
BC00540=948826
BC00541=948826
BC00542=970128
BC00543=961978
BC00544=961978
BC00545=951569
BC00546=840696
BC00547=518986
BC00548=509920
BC00549=467540
BC00550=467540
BC00551=467540
BC00552=521167
BC00553=520352
BC00554=535759
BC00555=535759
BC00556=535757
BC00557=535757
BC00558=535757
BC00559=535757
BC00560=485653
BC00561=485653
BC00562=485653
BC00563=485653
BC00564=485653
BC00565=485653
BC00566=485653
BC00567=485653
BC00568=485653
BC00569=485653
BC00570=485653
BC00571=600333
BC00572=615112
BC00573=615112
BC00574=615112
BC00575=615112
BC00576=615112
BC00577=615112
BC00578=615112
BC00579=615112
BC00580=615112
BC00581=615112
BC00582=615112
BC00583=615112
BC00584=615112
BC00585=615112
BC00586=658076
BC00587=658076
BC00588=658076
BC00589=658076
BC00590=655680
BC00591=656245
BC00592=762546
BC00593=762546
BC00594=799070
BC00595=799070
BC00596=799070
BC00597=799070
BC00598=799070
BC00599=799070
BC00600=799070
BC00601=799070
BC00602=799070
BC00603=799070
BC00604=799070
BC00605=799070
BC00606=799070
BC00607=845667
BC00608=845667
BC00609=845667
BC00610=845667
BC00611=845667
BC00612=969638
BC00613=930158
BC00614=945317
BC00615=945317
BC00616=945317
BC00617=945317
BC00618=945317
BC00619=946871
BC00620=945317
BC00621=945317
BC00622=945317
BC00623=937846
BC00624=907436
BC00625=895479
BC00626=639407
///POSTYPE BASE
///RECTAN
///RCONF 0,0,0,0,0,0,0,0,0,0,0,0,0,0,0,0,0,0,0,0,0,0,0,0
P00006=-2.449,0.031,8.825,0.0000,0.0000,0.0000
P00056=0.000,0.000,5.000,0.0000,0.0000,0.0000
P00301=0.005,-4.708,-4.628,0.0000,0.0000,0.0000
P00302=0.052,-2.937,-4.426,0.0000,0.0000,0.0000
P00303=-0.004,-1.437,-4.584,0.0000,0.0000,0.0000
P00304=0.028,-1.666,-4.234,0.0000,0.0000,0.0000
P00305=-0.003,-1.920,-3.501,0.0000,0.0000,0.0000
P00306=0.015,-2.252,-3.054,0.0000,0.0000,0.0000
P00307=0.019,-2.151,-5.077,0.0000,0.0000,0.0000
P00308=-0.003,-2.092,-4.888,0.0000,0.0000,0.0000
P00309=-0.040,-2.205,-4.992,0.0000,0.0000,0.0000
P00310=-0.006,-2.490,-5.925,0.0000,0.0000,0.0000
P00311=-0.007,-2.079,-5.307,0.0000,0.0000,0.0000
P00312=-0.032,2.202,-7.632,0.0000,0.0000,0.0000
P00351=13.563,-0.027,-0.653,0.0000,0.0000,0.0000
P00352=13.252,-0.027,-0.827,0.0000,0.0000,0.0000
P00353=10.971,-0.082,0.776,0.0000,0.0000,0.0000
P00354=-0.024,2.508,-1.824,0.0000,0.0000,0.0000
P00355=-0.001,2.528,-1.131,0.0000,0.0000,0.0000
P00356=-0.034,2.921,-0.262,0.0000,0.0000,0.0000
P00357=0.003,3.386,-0.091,0.0000,0.0000,0.0000
P00358=0.014,3.037,-0.020,0.0000,0.0000,0.0000
P00359=-0.005,2.731,0.912,0.0000,0.0000,0.0000
P00360=-0.011,3.412,0.438,0.0000,0.0000,0.0000
P00361=0.018,3.050,1.253,0.0000,0.0000,0.0000
P00362=0.014,2.784,0.148,0.0000,0.0000,0.0000
//INST
///DATE 2024/11/08 12:42
///ATTR SC,RW
///GROUP1 RB1,BS1
NOP
CALL JOB:MOVE_INTO_TUNNEL
MOVJ C00000 BC00000 VJ=10.00
MOVJ C00001 BC00001 VJ=10.00
MOVJ C00002 BC00002 VJ=10.00
MOVJ C00003 BC00003 VJ=10.00
MOVJ C00004 BC00004 VJ=10.00
'------------------------
'W29.2
'------------------------
MOVL C00005 BC00005 V=500.0
'------------------------
'W63.5
'------------------------
SFTOF
MOVL C00006 BC00006 V=166.7 PL=0
REFP 3 C00007 BC00007
CALL JOB:SEARCH-R1
IMOV P0056 V=50.0 PL=0
SET P0301 P0006
SFTON P0301
REFP 3 C00008 BC00008
CALL JOB:SEARCH-R1
SET P0301 P0006
SFTON P0301
MOVL C00009 BC00009 V=166.7 PL=0
SFTOF
MOVL C00010 BC00010 V=500.0
MOVL C00011 BC00011 V=166.7 PL=0
REFP 3 C00012 BC00012
CALL JOB:SEARCH-R1
IMOV P0056 V=50.0 PL=0
SET P0302 P0006
SFTON P0302
REFP 3 C00013 BC00013
CALL JOB:SEARCH-R1
SET P0302 P0006
SFTON P0302
MOVL C00014 BC00014 V=166.7 PL=0
SFTOF
MOVL C00015 BC00015 V=500.0
MOVL C00016 BC00016 V=166.7 PL=0
REFP 3 C00017 BC00017
CALL JOB:SEARCH-R1
IMOV P0056 V=50.0 PL=0
SET P0303 P0006
SFTON P0303
REFP 3 C00018 BC00018
CALL JOB:SEARCH-R1
SET P0303 P0006
SFTON P0303
SFTOF
MOVL C00019 BC00019 V=166.7 PL=0
MOVL C00020 BC00020 V=500.0
MOVJ C00021 BC00021 VJ=30.00
MOVJ C00022 BC00022 VJ=30.00
MOVJ C00023 BC00023 VJ=30.00
MOVL C00024 BC00024 V=500.0
'------------------------
'W29.14
'------------------------
MOVL C00025 BC00025 V=166.7 PL=0
REFP 3 C00026 BC00026
CALL JOB:SEARCH-R1
IMOV P0056 V=23.0 PL=0
SET P0304 P0006
SFTON P0304
REFP 3 C00027 BC00027
CALL JOB:SEARCH-R1
SET P0304 P0006
SFTON P0304
MOVL C00028 BC00028 V=66.7 PL=0
SFTOF
'PRZEJAZD
MOVL C00029 BC00029 V=500.0
MOVL C00030 BC00030 V=500.0
'------------------------
'W63.17
'------------------------
MOVL C00031 BC00031 V=166.7 PL=0
REFP 3 C00032 BC00032
CALL JOB:SEARCH-R1
IMOV P0056 V=23.0 PL=0
SET P0305 P0006
SFTON P0305
REFP 3 C00033 BC00033
CALL JOB:SEARCH-R1
SET P0305 P0006
SFTON P0305
MOVL C00034 BC00034 V=166.7 PL=0
SFTOF
MOVL C00035 BC00035 V=500.0
MOVL C00036 BC00036 V=166.7
REFP 3 C00037 BC00037
CALL JOB:SEARCH-R1
IMOV P0056 V=23.0 PL=0
SET P0306 P0006
SFTON P0306
REFP 3 C00038 BC00038
CALL JOB:SEARCH-R1
SET P0306 P0006
SFTON P0306
MOVL C00039 BC00039 V=166.7 PL=0
'PRZEJAZD
MOVL C00040 BC00040 V=500.0
MOVL C00041 BC00041 V=166.7
REFP 3 C00042 BC00042
CALL JOB:SEARCH-R1
IMOV P0056 V=23.0 PL=0
SET P0307 P0006
SFTON P0307
REFP 3 C00043 BC00043
CALL JOB:SEARCH-R1
SET P0307 P0006
SFTON P0307
MOVL C00044 BC00044 V=166.7 PL=0
SFTOF
MOVJ C00045 BC00045 VJ=20.00
MOVJ C00046 BC00046 VJ=20.00
MOVJ C00047 BC00047 VJ=30.00
MOVJ C00048 BC00048 VJ=30.00
MOVJ C00049 BC00049 VJ=30.00
MOVL C00050 BC00050 V=500.0
'------------------------
'W63.20
'------------------------
MOVL C00051 BC00051 V=166.7 PL=0
REFP 3 C00052 BC00052
CALL JOB:SEARCH-R1
IMOV P0056 V=23.0 PL=0
SET P0308 P0006
SFTON P0308
REFP 3 C00053 BC00053
CALL JOB:SEARCH-R1
SET P0308 P0006
SFTON P0308
MOVL C00054 BC00054 V=166.7 PL=0
SFTOF
'PRZEJAZD
MOVL C00055 BC00055 V=500.0
'------------------------
'W63.23
'------------------------
MOVL C00056 BC00056 V=166.7 PL=0
REFP 3 C00057 BC00057
CALL JOB:SEARCH-R1
IMOV P0056 V=23.0 PL=0
SET P0309 P0006
SFTON P0309
REFP 3 C00058 BC00058
CALL JOB:SEARCH-R1
SET P0309 P0006
SFTON P0309
MOVL C00059 BC00059 V=250.0 PL=0
SFTOF
MOVL C00060 BC00060 V=500.0
MOVL C00061 BC00061 V=166.7 PL=0
REFP 3 C00062 BC00062
CALL JOB:SEARCH-R1
IMOV P0056 V=23.0 PL=0
SET P0310 P0006
SFTON P0310
REFP 3 C00063 BC00063
CALL JOB:SEARCH-R1
SET P0310 P0006
SFTON P0310
MOVL C00064 BC00064 V=250.0 PL=0
SFTOF
MOVL C00065 BC00065 V=500.0
MOVL C00066 BC00066 V=166.7 PL=0
REFP 3 C00067 BC00067
CALL JOB:SEARCH-R1
IMOV P0056 V=23.0 PL=0
SET P0311 P0006
SFTON P0311
REFP 3 C00068 BC00068
CALL JOB:SEARCH-R1
SET P0311 P0006
SFTON P0311
MOVL C00069 BC00069 V=250.0 PL=0
SFTOF
MOVL C00070 BC00070 V=500.0
MOVL C00071 BC00071 V=500.0
MOVL C00072 BC00072 V=333.3
'------------------------
'W29.29
'------------------------
MOVL C00073 BC00073 V=166.7 PL=0
REFP 3 C00074 BC00074
CALL JOB:SEARCH-R1
IMOV P0056 V=23.0 PL=0
SET P0312 P0006
SFTON P0312
REFP 3 C00075 BC00075
CALL JOB:SEARCH-R1
SET P0312 P0006
SFTON P0312
MOVL C00076 BC00076 V=250.0 PL=0
SFTOF
'PRZEJAZD
MOVL C00077 BC00077 V=333.3
'PRZEJAZD
MOVJ C00078 BC00078 VJ=30.00
MOVJ C00079 BC00079 VJ=20.00
MOVJ C00080 BC00080 VJ=50.00
MOVJ C00081 BC00081 VJ=20.00
MOVJ C00082 BC00082 VJ=10.00
MOVJ C00083 BC00083 VJ=20.00
MOVJ C00084 BC00084 VJ=20.00
'------------------------
'W28.2
'------------------------
MOVJ C00085 BC00085 VJ=10.00
MOVJ C00086 BC00086 VJ=10.00
MOVL C00087 BC00087 V=500.0
MOVL C00088 BC00088 V=500.0
'------------------------
'W62.5
'------------------------
MOVL C00089 BC00089 V=166.7 PL=0
REFP 3 C00090 BC00090
CALL JOB:SEARCH-R1
IMOV P0056 V=23.0 PL=0
SET P0351 P0006
SFTON P0351
REFP 3 C00091 BC00091
CALL JOB:SEARCH-R1
SET P0351 P0006
SFTON P0351
MOVL C00092 BC00092 V=250.0 PL=0
SFTOF
'PRZEJAZD
MOVL C00093 BC00093 V=500.0
MOVL C00094 BC00094 V=500.0
MOVL C00095 BC00095 V=500.0
MOVL C00096 BC00096 V=166.7 PL=0
REFP 3 C00097 BC00097
CALL JOB:SEARCH-R1
IMOV P0056 V=23.0 PL=0
SET P0352 P0006
SFTON P0352
REFP 3 C00098 BC00098
CALL JOB:SEARCH-R1
SET P0352 P0006
SFTON P0352
MOVL C00099 BC00099 V=250.0 PL=0
SFTOF
MOVL C00100 BC00100 V=500.0
'------------------------
'W29.8
'------------------------
MOVL C00101 BC00101 V=166.7 PL=0
REFP 3 C00102 BC00102
CALL JOB:SEARCH-R1
IMOV P0056 V=23.0 PL=0
SET P0353 P0006
SFTON P0353
REFP 3 C00103 BC00103
CALL JOB:SEARCH-R1
SET P0353 P0006
SFTON P0353
MOVL C00104 BC00104 V=250.0 PL=0
SFTOF
MOVL C00105 BC00105 V=500.0
'PRZEJAZD
MOVL C00106 BC00106 V=500.0
MOVJ C00107 BC00107 VJ=20.00
MOVL C00108 BC00108 V=500.0
MOVL C00109 BC00109 V=500.0
MOVL C00110 BC00110 V=500.0
'------------------------
'W29.11
'------------------------
MOVL C00111 BC00111 V=166.7 PL=0
REFP 3 C00112 BC00112
CALL JOB:SEARCH-R1
IMOV P0056 V=23.0 PL=0
SET P0354 P0006
SFTON P0354
REFP 3 C00113 BC00113
CALL JOB:SEARCH-R1
SET P0354 P0006
SFTON P0354
MOVL C00114 BC00114 V=250.0 PL=0
SFTOF
'PRZEJAZD
MOVL C00115 BC00115 V=500.0
'------------------------
'W29.14
'------------------------
MOVL C00116 BC00116 V=166.7 PL=0
REFP 3 C00117 BC00117
CALL JOB:SEARCH-R1
IMOV P0056 V=23.0 PL=0
SET P0355 P0006
SFTON P0355
REFP 3 C00118 BC00118
CALL JOB:SEARCH-R1
SET P0355 P0006
SFTON P0355
MOVL C00119 BC00119 V=250.0 PL=0
SFTOF
'PRZEJAZD
MOVL C00120 BC00120 V=500.0
'------------------------
'W63.17
'------------------------
MOVL C00121 BC00121 V=166.7 PL=0
REFP 3 C00122 BC00122
CALL JOB:SEARCH-R1
IMOV P0056 V=23.0 PL=0
SET P0356 P0006
SFTON P0356
REFP 3 C00123 BC00123
CALL JOB:SEARCH-R1
SET P0356 P0006
SFTON P0356
MOVL C00124 BC00124 V=250.0 PL=0
SFTOF
MOVL C00125 BC00125 V=500.0
MOVL C00126 BC00126 V=166.7 PL=0
REFP 3 C00127 BC00127
CALL JOB:SEARCH-R1
IMOV P0056 V=23.0 PL=0
SET P0357 P0006
SFTON P0357
REFP 3 C00128 BC00128
CALL JOB:SEARCH-R1
SET P0357 P0006
SFTON P0357
MOVL C00129 BC00129 V=250.0 PL=0
SFTOF
'PRZEJAZD
MOVL C00130 BC00130 V=500.0
MOVJ C00131 BC00131 VJ=30.00
MOVJ C00132 BC00132 VJ=30.00
MOVJ C00133 BC00133 VJ=30.00
MOVL C00134 BC00134 V=500.0
MOVL C00135 BC00135 V=500.0
'------------------------
'W62.20
'------------------------
MOVL C00136 BC00136 V=166.7 PL=0
REFP 3 C00137 BC00137
CALL JOB:SEARCH-R1
IMOV P0056 V=23.0 PL=0
SET P0358 P0006
SFTON P0358
REFP 3 C00138 BC00138
CALL JOB:SEARCH-R1
SET P0358 P0006
SFTON P0358
MOVL C00139 BC00139 V=250.0 PL=0
SFTOF
'PRZEJAZD
MOVL C00140 BC00140 V=500.0
'------------------------
'W63.23
'------------------------
MOVL C00141 BC00141 V=166.7 PL=0
REFP 3 C00142 BC00142
CALL JOB:SEARCH-R1
IMOV P0056 V=23.0 PL=0
SET P0359 P0006
SFTON P0359
REFP 3 C00143 BC00143
CALL JOB:SEARCH-R1
SET P0359 P0006
SFTON P0359
MOVL C00144 BC00144 V=250.0 PL=0
MOVL C00145 BC00145 V=500.0
'------------------------
'W29.29
'------------------------
MOVL C00146 BC00146 V=166.7 PL=0
REFP 3 C00147 BC00147
CALL JOB:SEARCH-R1
IMOV P0056 V=23.0 PL=0
SET P0360 P0006
SFTON P0360
REFP 3 C00148 BC00148
CALL JOB:SEARCH-R1
SET P0360 P0006
SFTON P0360
MOVL C00149 BC00149 V=250.0 PL=0
SFTOF
'PRZEJAZD
MOVL C00150 BC00150 V=500.0
MOVL C00151 BC00151 V=166.7 PL=0
REFP 3 C00152 BC00152
CALL JOB:SEARCH-R1
IMOV P0056 V=23.0 PL=0
SET P0361 P0006
SFTON P0361
REFP 3 C00153 BC00153
CALL JOB:SEARCH-R1
SET P0361 P0006
SFTON P0361
MOVL C00154 BC00154 V=250.0 PL=0
SFTOF
'------------------------
'W29.32
'------------------------
'PRZEJAZD
MOVL C00155 BC00155 V=500.0
MOVJ C00156 BC00156 VJ=10.00
MOVL C00157 BC00157 V=416.7
MOVL C00158 BC00158 V=166.7 PL=0
REFP 3 C00159 BC00159
CALL JOB:SEARCH-R1
IMOV P0056 V=23.0 PL=0
SET P0362 P0006
SFTON P0362
REFP 3 C00160 BC00160
CALL JOB:SEARCH-R1
SET P0362 P0006
SFTON P0362
MOVL C00161 BC00161 V=250.0 PL=0
SFTOF
MOVJ C00162 BC00162 VJ=20.00
MOVJ C00163 BC00163 VJ=30.00
MOVJ C00164 BC00164 VJ=30.00
'KONIEC SEARCH WEW STRONA
MOVJ C00165 BC00165 VJ=30.00
MOVJ C00166 BC00166 VJ=20.00
MOVJ C00167 BC00167 VJ=10.00
MOVJ C00168 BC00168 VJ=20.00
MOVJ C00169 BC00169 VJ=20.00
'------------------------
'W29.2
'------------------------
MOVL C00170 BC00170 V=500.0
'------------------------
'W63.5
MACRO1 MJ#(0) ARGF9
'------------------------
SFTOF
SFTON P0301
MOVL C00171 BC00171 V=166.7 PL=0
ARCON
MOVL C00172 BC00172 V=10.0
ARCOF
SFTOF
MOVL C00173 BC00173 V=500.0
SFTON P0302
MOVL C00174 BC00174 V=166.7 PL=0
ARCON
MOVL C00175 BC00175 V=10.0
ARCOF
MOVL C00176 BC00176 V=166.7 PL=0
SFTOF
MOVL C00177 BC00177 V=500.0
SFTON P0303
MOVL C00178 BC00178 V=166.7 PL=0
ARCON
MOVL C00179 BC00179 V=10.0
ARCOF
SFTOF
MOVL C00180 BC00180 V=166.7 PL=0
MOVL C00181 BC00181 V=500.0
MOVJ C00182 BC00182 VJ=30.00
MOVJ C00183 BC00183 VJ=30.00
MOVJ C00184 BC00184 VJ=30.00
MOVL C00185 BC00185 V=500.0
'------------------------
'W29.14
'------------------------
SFTON P0304
MOVL C00186 BC00186 V=166.7 PL=0
ARCON
MOVL C00187 BC00187 V=10.0
ARCOF
MOVL C00188 BC00188 V=166.7 PL=0
SFTOF
'PRZEJAZD
MOVL C00189 BC00189 V=500.0
MOVL C00190 BC00190 V=500.0
'------------------------
'W63.17
'------------------------
SFTON P0305
MOVL C00191 BC00191 V=166.7 PL=0
ARCON
MOVL C00192 BC00192 V=10.0
ARCOF
MOVL C00193 BC00193 V=166.7 PL=0
SFTOF
MOVL C00194 BC00194 V=500.0
SFTON P0306
MOVL C00195 BC00195 V=166.7
ARCON
MOVL C00196 BC00196 V=10.0
ARCOF
MOVL C00197 BC00197 V=166.7 PL=0
SFTOF
'PRZEJAZD
MOVL C00198 BC00198 V=500.0
SFTON P0307
MOVL C00199 BC00199 V=166.7
ARCON
MOVL C00200 BC00200 V=10.0
ARCOF
MOVL C00201 BC00201 V=166.7 PL=0
SFTOF
MOVJ C00202 BC00202 VJ=20.00
MOVJ C00203 BC00203 VJ=20.00
MOVJ C00204 BC00204 VJ=30.00
MOVJ C00205 BC00205 VJ=30.00
MOVJ C00206 BC00206 VJ=30.00
MOVL C00207 BC00207 V=500.0
'------------------------
'W63.20
'------------------------
SFTON P0308
MOVL C00208 BC00208 V=166.7 PL=0
ARCON
MOVL C00209 BC00209 V=10.0
ARCOF
MOVL C00210 BC00210 V=166.7 PL=0
SFTOF
'PRZEJAZD
MOVL C00211 BC00211 V=500.0
'------------------------
'W63.23
'------------------------
SFTON P0309
MOVL C00212 BC00212 V=166.7 PL=0
ARCON
MOVL C00213 BC00213 V=10.0
ARCOF
MOVL C00214 BC00214 V=250.0 PL=0
SFTOF
MOVL C00215 BC00215 V=500.0
SFTON P0310
MOVL C00216 BC00216 V=166.7 PL=0
ARCON
MOVL C00217 BC00217 V=10.0
ARCOF
MOVL C00218 BC00218 V=250.0 PL=0
SFTOF
MOVL C00219 BC00219 V=500.0
SFTON P0311
MOVL C00220 BC00220 V=166.7 PL=0
ARCON
MOVL C00221 BC00221 V=10.0
ARCOF
MOVL C00222 BC00222 V=250.0 PL=0
SFTOF
MOVL C00223 BC00223 V=500.0
MOVL C00224 BC00224 V=500.0
MOVL C00225 BC00225 V=333.3
COMM MOVL C00226 BC00226 V=250.0
'------------------------
'W29.29
'------------------------
SFTON P0312
COMM MOVL C00227 BC00227 V=166.7 PL=0
COMM ARCON
COMM MOVL C00228 BC00228 V=9.2
COMM ARCOF
COMM MOVL C00229 BC00229 V=250.0 PL=0
MOVL C00230 BC00230 V=333.3
ARCON
MOVL C00231 BC00231 V=9.2
ARCOF
SFTOF
'PRZEJAZD
MOVL C00232 BC00232 V=333.3
MOVJ C00233 BC00233 VJ=30.00
MOVJ C00234 BC00234 VJ=20.00
MOVJ C00235 BC00235 VJ=50.00
MOVJ C00236 BC00236 VJ=20.00
MOVJ C00237 BC00237 VJ=10.00
MOVJ C00238 BC00238 VJ=20.00
MOVJ C00239 BC00239 VJ=20.00
'------------------------
'W28.2
'------------------------
MOVJ C00240 BC00240 VJ=10.00
MOVJ C00241 BC00241 VJ=10.00
MOVL C00242 BC00242 V=500.0
MOVL C00243 BC00243 V=500.0
'------------------------
'W62.5
'------------------------
SFTON P0351
MOVL C00244 BC00244 V=166.7 PL=0
ARCON
MOVL C00245 BC00245 V=10.0
ARCOF
MOVL C00246 BC00246 V=250.0 PL=0
SFTOF
'PRZEJAZD
MOVL C00247 BC00247 V=500.0
MOVL C00248 BC00248 V=500.0
MOVL C00249 BC00249 V=500.0
SFTON P0352
MOVL C00250 BC00250 V=166.7 PL=0
ARCON
MOVL C00251 BC00251 V=10.0
ARCOF
MOVL C00252 BC00252 V=250.0 PL=0
SFTOF
MOVL C00253 BC00253 V=500.0
'------------------------
'W29.8
'------------------------
SFTON P0353
MOVL C00254 BC00254 V=166.7 PL=0
ARCON
MOVL C00255 BC00255 V=10.0
ARCOF
MOVL C00256 BC00256 V=250.0 PL=0
SFTOF
MOVL C00257 BC00257 V=500.0
'PRZEJAZD
MOVL C00258 BC00258 V=500.0
MOVJ C00259 BC00259 VJ=20.00
MOVL C00260 BC00260 V=500.0
MOVL C00261 BC00261 V=500.0
MOVL C00262 BC00262 V=500.0
'------------------------
'W29.11
'------------------------
SFTON P0354
MOVL C00263 BC00263 V=166.7 PL=0
ARCON
MOVL C00264 BC00264 V=10.0
ARCOF
MOVL C00265 BC00265 V=250.0 PL=0
SFTOF
'PRZEJAZD
MOVL C00266 BC00266 V=500.0
'------------------------
'W29.14
'------------------------
SFTON P0355
MOVL C00267 BC00267 V=166.7 PL=0
ARCON
MOVL C00268 BC00268 V=10.0
ARCOF
MOVL C00269 BC00269 V=250.0 PL=0
SFTOF
'PRZEJAZD
MOVL C00270 BC00270 V=500.0
'------------------------
'W63.17
'------------------------
SFTON P0356
MOVL C00271 BC00271 V=166.7 PL=0
ARCON
MOVL C00272 BC00272 V=10.0
ARCOF
MOVL C00273 BC00273 V=250.0 PL=0
SFTOF
MOVL C00274 BC00274 V=500.0
SFTON P0357
MOVL C00275 BC00275 V=166.7 PL=0
ARCON
MOVL C00276 BC00276 V=10.0
ARCOF
MOVL C00277 BC00277 V=250.0 PL=0
SFTOF
'PRZEJAZD
MOVL C00278 BC00278 V=500.0
MOVJ C00279 BC00279 VJ=30.00
MOVJ C00280 BC00280 VJ=30.00
MOVJ C00281 BC00281 VJ=30.00
MOVL C00282 BC00282 V=500.0
MOVL C00283 BC00283 V=500.0
'------------------------
'W62.20
'------------------------
SFTON P0358
MOVL C00284 BC00284 V=166.7 PL=0
ARCON
MOVL C00285 BC00285 V=10.0
ARCOF
MOVL C00286 BC00286 V=250.0 PL=0
SFTOF
'PRZEJAZD
MOVL C00287 BC00287 V=500.0
'------------------------
'W63.23
'------------------------
SFTON P0359
MOVL C00288 BC00288 V=166.7 PL=0
ARCON
MOVL C00289 BC00289 V=10.0
ARCOF
MOVL C00290 BC00290 V=250.0 PL=0
MOVL C00291 BC00291 V=500.0
'------------------------
'W29.29
'------------------------
SFTON P0360
MOVL C00292 BC00292 V=166.7 PL=0
ARCON
MOVL C00293 BC00293 V=10.0
ARCOF
MOVL C00294 BC00294 V=250.0 PL=0
SFTOF
'PRZEJAZD
MOVL C00295 BC00295 V=500.0
SFTON P0361
MOVL C00296 BC00296 V=166.7 PL=0
ARCON
MOVL C00297 BC00297 V=10.0
ARCOF
MOVL C00298 BC00298 V=250.0 PL=0
SFTOF
'------------------------
'W29.32
'------------------------
'PRZEJAZD
MOVL C00299 BC00299 V=500.0
MOVJ C00300 BC00300 VJ=10.00
COMM MOVL C00301 BC00301 V=416.7
COMM SFTON P0362
COMM MOVL C00302 BC00302 V=166.7 PL=0
COMM ARCON
COMM MOVL C00303 BC00303 V=9.2
COMM ARCOF
COMM MOVL C00304 BC00304 V=250.0 PL=0
COMM MOVL C00305 BC00305 V=250.0
SFTON P0362
MOVL C00306 BC00306 V=166.7
ARCON
MOVL C00307 BC00307 V=9.2
ARCOF
SFTOF
MOVL C00308 BC00308 V=166.7
MOVJ C00309 BC00309 VJ=20.00
MOVJ C00310 BC00310 VJ=30.00
MOVJ C00311 BC00311 VJ=30.00
CALL JOB:MOVE_OUT_OF_TUNNEL
CALL JOB:CLEAN-R1
CALL JOB:MOVE_INTO_TUNNEL
'KONIEC SPAWANIA WEW STRONA
MOVJ C00312 BC00312 VJ=10.00
MOVJ C00313 BC00313 VJ=10.00
MOVJ C00314 BC00314 VJ=20.00
MOVJ C00315 BC00315 VJ=20.00
MOVJ C00316 BC00316 VJ=10.00
MOVJ C00317 BC00317 VJ=10.00
'------------------------
'W29.2
'------------------------
MOVL C00318 BC00318 V=500.0
'------------------------
'W63.5
'------------------------
SFTOF
MOVL C00319 BC00319 V=166.7 PL=0
REFP 3 C00320 BC00320
CALL JOB:SEARCH-R1
IMOV P0056 V=50.0 PL=0
SET P0301 P0006
SFTON P0301
REFP 3 C00321 BC00321
CALL JOB:SEARCH-R1
SET P0301 P0006
SFTON P0301
MOVL C00322 BC00322 V=166.7 PL=0
SFTOF
MOVL C00323 BC00323 V=500.0
MOVL C00324 BC00324 V=166.7 PL=0
REFP 3 C00325 BC00325
CALL JOB:SEARCH-R1
IMOV P0056 V=50.0 PL=0
SET P0302 P0006
SFTON P0302
REFP 3 C00326 BC00326
CALL JOB:SEARCH-R1
SET P0302 P0006
SFTON P0302
MOVL C00327 BC00327 V=166.7 PL=0
SFTOF
MOVL C00328 BC00328 V=500.0
MOVL C00329 BC00329 V=166.7 PL=0
REFP 3 C00330 BC00330
CALL JOB:SEARCH-R1
IMOV P0056 V=50.0 PL=0
SET P0303 P0006
SFTON P0303
REFP 3 C00331 BC00331
CALL JOB:SEARCH-R1
SET P0303 P0006
SFTON P0303
SFTOF
MOVL C00332 BC00332 V=166.7 PL=0
MOVL C00333 BC00333 V=500.0
MOVJ C00334 BC00334 VJ=30.00
MOVJ C00335 BC00335 VJ=30.00
MOVJ C00336 BC00336 VJ=20.00
MOVJ C00337 BC00337 VJ=30.00
MOVL C00338 BC00338 V=500.0
'------------------------
'W29.14
'------------------------
MOVL C00339 BC00339 V=166.7 PL=0
REFP 3 C00340 BC00340
CALL JOB:SEARCH-R1
IMOV P0056 V=23.0 PL=0
SET P0304 P0006
SFTON P0304
REFP 3 C00341 BC00341
CALL JOB:SEARCH-R1
SET P0304 P0006
SFTON P0304
MOVL C00342 BC00342 V=66.7 PL=0
SFTOF
'PRZEJAZD
MOVL C00343 BC00343 V=500.0
MOVL C00344 BC00344 V=500.0
'------------------------
'W63.17
'------------------------
MOVL C00345 BC00345 V=166.7 PL=0
REFP 3 C00346 BC00346
CALL JOB:SEARCH-R1
IMOV P0056 V=23.0 PL=0
SET P0305 P0006
SFTON P0305
REFP 3 C00347 BC00347
CALL JOB:SEARCH-R1
SET P0305 P0006
SFTON P0305
MOVL C00348 BC00348 V=166.7 PL=0
SFTOF
MOVL C00349 BC00349 V=500.0
MOVL C00350 BC00350 V=166.7
REFP 3 C00351 BC00351
CALL JOB:SEARCH-R1
IMOV P0056 V=23.0 PL=0
SET P0306 P0006
SFTON P0306
REFP 3 C00352 BC00352
CALL JOB:SEARCH-R1
SET P0306 P0006
SFTON P0306
MOVL C00353 BC00353 V=166.7 PL=0
'PRZEJAZD
MOVL C00354 BC00354 V=500.0
MOVL C00355 BC00355 V=166.7
REFP 3 C00356 BC00356
CALL JOB:SEARCH-R1
IMOV P0056 V=23.0 PL=0
SET P0307 P0006
SFTON P0307
REFP 3 C00357 BC00357
CALL JOB:SEARCH-R1
SET P0307 P0006
SFTON P0307
MOVL C00358 BC00358 V=166.7 PL=0
SFTOF
MOVJ C00359 BC00359 VJ=20.00
MOVJ C00360 BC00360 VJ=20.00
MOVJ C00361 BC00361 VJ=30.00
MOVJ C00362 BC00362 VJ=30.00
MOVL C00363 BC00363 V=500.0
'------------------------
'W63.20
'------------------------
MOVL C00364 BC00364 V=166.7 PL=0
REFP 3 C00365 BC00365
CALL JOB:SEARCH-R1
IMOV P0056 V=23.0 PL=0
SET P0308 P0006
SFTON P0308
REFP 3 C00366 BC00366
CALL JOB:SEARCH-R1
SET P0308 P0006
SFTON P0308
MOVL C00367 BC00367 V=166.7 PL=0
SFTOF
'PRZEJAZD
MOVL C00368 BC00368 V=500.0
'------------------------
'W63.23
'------------------------
MOVL C00369 BC00369 V=166.7 PL=0
REFP 3 C00370 BC00370
CALL JOB:SEARCH-R1
IMOV P0056 V=23.0 PL=0
SET P0309 P0006
SFTON P0309
REFP 3 C00371 BC00371
CALL JOB:SEARCH-R1
SET P0309 P0006
SFTON P0309
MOVL C00372 BC00372 V=250.0 PL=0
SFTOF
MOVL C00373 BC00373 V=500.0
MOVL C00374 BC00374 V=166.7 PL=0
REFP 3 C00375 BC00375
CALL JOB:SEARCH-R1
IMOV P0056 V=23.0 PL=0
SET P0310 P0006
SFTON P0310
REFP 3 C00376 BC00376
CALL JOB:SEARCH-R1
SET P0310 P0006
SFTON P0310
MOVL C00377 BC00377 V=250.0 PL=0
SFTOF
MOVL C00378 BC00378 V=500.0
MOVL C00379 BC00379 V=166.7 PL=0
REFP 3 C00380 BC00380
CALL JOB:SEARCH-R1
IMOV P0056 V=23.0 PL=0
SET P0311 P0006
SFTON P0311
REFP 3 C00381 BC00381
CALL JOB:SEARCH-R1
SET P0311 P0006
SFTON P0311
MOVL C00382 BC00382 V=250.0 PL=0
SFTOF
MOVL C00383 BC00383 V=500.0
MOVL C00384 BC00384 V=500.0
MOVL C00385 BC00385 V=333.3
'------------------------
'W29.29
'------------------------
MOVL C00386 BC00386 V=250.0
MOVL C00387 BC00387 V=166.7 PL=0
REFP 3 C00388 BC00388
CALL JOB:SEARCH-R1
IMOV P0056 V=23.0 PL=0
SET P0312 P0006
SFTON P0312
REFP 3 C00389 BC00389
CALL JOB:SEARCH-R1
SET P0312 P0006
SFTON P0312
MOVL C00390 BC00390 V=250.0 PL=0
SFTOF
'PRZEJAZD
MOVL C00391 BC00391 V=333.3
'PRZEJAZD
MOVJ C00392 BC00392 VJ=20.00
MOVJ C00393 BC00393 VJ=50.00
MOVJ C00394 BC00394 VJ=20.00
MOVJ C00395 BC00395 VJ=10.00
'------------------------
'W28.2
'------------------------
MOVJ C00396 BC00396 VJ=10.00
MOVJ C00397 BC00397 VJ=10.00
MOVL C00398 BC00398 V=500.0
MOVL C00399 BC00399 V=500.0
'------------------------
'W62.5
'------------------------
MOVL C00400 BC00400 V=166.7 PL=0
REFP 3 C00401 BC00401
CALL JOB:SEARCH-R1
IMOV P0056 V=23.0 PL=0
SET P0351 P0006
SFTON P0351
REFP 3 C00402 BC00402
CALL JOB:SEARCH-R1
SET P0351 P0006
SFTON P0351
MOVL C00403 BC00403 V=250.0 PL=0
SFTOF
'PRZEJAZD
MOVL C00404 BC00404 V=500.0
MOVL C00405 BC00405 V=500.0
MOVL C00406 BC00406 V=500.0
MOVL C00407 BC00407 V=166.7 PL=0
REFP 3 C00408 BC00408
CALL JOB:SEARCH-R1
IMOV P0056 V=23.0 PL=0
SET P0352 P0006
SFTON P0352
REFP 3 C00409 BC00409
CALL JOB:SEARCH-R1
SET P0352 P0006
SFTON P0352
MOVL C00410 BC00410 V=250.0 PL=0
SFTOF
MOVL C00411 BC00411 V=500.0
'------------------------
'W29.8
'------------------------
MOVL C00412 BC00412 V=166.7 PL=0
REFP 3 C00413 BC00413
CALL JOB:SEARCH-R1
IMOV P0056 V=23.0 PL=0
SET P0353 P0006
SFTON P0353
REFP 3 C00414 BC00414
CALL JOB:SEARCH-R1
SET P0353 P0006
SFTON P0353
MOVL C00415 BC00415 V=250.0 PL=0
SFTOF
MOVL C00416 BC00416 V=500.0
'PRZEJAZD
MOVL C00417 BC00417 V=500.0
MOVJ C00418 BC00418 VJ=20.00
MOVJ C00419 BC00419 VJ=20.00
MOVL C00420 BC00420 V=500.0
MOVL C00421 BC00421 V=500.0
MOVL C00422 BC00422 V=500.0
'------------------------
'W29.11
'------------------------
MOVL C00423 BC00423 V=166.7 PL=0
REFP 3 C00424 BC00424
CALL JOB:SEARCH-R1
IMOV P0056 V=23.0 PL=0
SET P0354 P0006
SFTON P0354
REFP 3 C00425 BC00425
CALL JOB:SEARCH-R1
SET P0354 P0006
SFTON P0354
MOVL C00426 BC00426 V=250.0 PL=0
SFTOF
'PRZEJAZD
MOVL C00427 BC00427 V=500.0
'------------------------
'W29.14
'------------------------
MOVL C00428 BC00428 V=166.7 PL=0
REFP 3 C00429 BC00429
CALL JOB:SEARCH-R1
IMOV P0056 V=23.0 PL=0
SET P0355 P0006
SFTON P0355
REFP 3 C00430 BC00430
CALL JOB:SEARCH-R1
SET P0355 P0006
SFTON P0355
MOVL C00431 BC00431 V=250.0 PL=0
SFTOF
'PRZEJAZD
MOVL C00432 BC00432 V=500.0
'------------------------
'W63.17
'------------------------
MOVL C00433 BC00433 V=166.7 PL=0
REFP 3 C00434 BC00434
CALL JOB:SEARCH-R1
IMOV P0056 V=23.0 PL=0
SET P0356 P0006
SFTON P0356
REFP 3 C00435 BC00435
CALL JOB:SEARCH-R1
SET P0356 P0006
SFTON P0356
MOVL C00436 BC00436 V=250.0 PL=0
SFTOF
MOVL C00437 BC00437 V=500.0
MOVL C00438 BC00438 V=166.7 PL=0
REFP 3 C00439 BC00439
CALL JOB:SEARCH-R1
IMOV P0056 V=23.0 PL=0
SET P0357 P0006
SFTON P0357
REFP 3 C00440 BC00440
CALL JOB:SEARCH-R1
SET P0357 P0006
SFTON P0357
MOVL C00441 BC00441 V=250.0 PL=0
SFTOF
'PRZEJAZD
MOVL C00442 BC00442 V=500.0
MOVJ C00443 BC00443 VJ=30.00
MOVJ C00444 BC00444 VJ=30.00
MOVL C00445 BC00445 V=500.0
MOVL C00446 BC00446 V=500.0
'------------------------
'W62.20
'------------------------
MOVL C00447 BC00447 V=166.7 PL=0
REFP 3 C00448 BC00448
CALL JOB:SEARCH-R1
IMOV P0056 V=23.0 PL=0
SET P0358 P0006
SFTON P0358
REFP 3 C00449 BC00449
CALL JOB:SEARCH-R1
SET P0358 P0006
SFTON P0358
MOVL C00450 BC00450 V=250.0 PL=0
SFTOF
'PRZEJAZD
MOVL C00451 BC00451 V=500.0
'------------------------
'W63.23
'------------------------
MOVL C00452 BC00452 V=166.7 PL=0
REFP 3 C00453 BC00453
CALL JOB:SEARCH-R1
IMOV P0056 V=23.0 PL=0
SET P0359 P0006
SFTON P0359
REFP 3 C00454 BC00454
CALL JOB:SEARCH-R1
SET P0359 P0006
SFTON P0359
MOVL C00455 BC00455 V=250.0 PL=0
MOVL C00456 BC00456 V=500.0
'------------------------
'W29.29
'------------------------
MOVL C00457 BC00457 V=166.7 PL=0
REFP 3 C00458 BC00458
CALL JOB:SEARCH-R1
IMOV P0056 V=23.0 PL=0
SET P0360 P0006
SFTON P0360
REFP 3 C00459 BC00459
CALL JOB:SEARCH-R1
SET P0360 P0006
SFTON P0360
MOVL C00460 BC00460 V=250.0 PL=0
SFTOF
'PRZEJAZD
MOVL C00461 BC00461 V=500.0
MOVL C00462 BC00462 V=166.7 PL=0
REFP 3 C00463 BC00463
CALL JOB:SEARCH-R1
IMOV P0056 V=23.0 PL=0
SET P0361 P0006
SFTON P0361
REFP 3 C00464 BC00464
CALL JOB:SEARCH-R1
SET P0361 P0006
SFTON P0361
MOVL C00465 BC00465 V=250.0 PL=0
SFTOF
'------------------------
'W29.32
'------------------------
'PRZEJAZD
MOVL C00466 BC00466 V=500.0
MOVL C00467 BC00467 V=500.0
MOVL C00468 BC00468 V=416.7
MOVL C00469 BC00469 V=166.7 PL=0
REFP 3 C00470 BC00470
CALL JOB:SEARCH-R1
IMOV P0056 V=23.0 PL=0
SET P0362 P0006
SFTON P0362
REFP 3 C00471 BC00471
CALL JOB:SEARCH-R1
SET P0362 P0006
SFTON P0362
MOVL C00472 BC00472 V=250.0 PL=0
SFTOF
MOVJ C00473 BC00473 VJ=20.00
MOVJ C00474 BC00474 VJ=30.00
MOVJ C00475 BC00475 VJ=30.00
'KONIEC SEARCH WEW STRONA
MOVJ C00476 BC00476 VJ=30.00
MOVJ C00477 BC00477 VJ=20.00
MOVJ C00478 BC00478 VJ=10.00
MOVJ C00479 BC00479 VJ=20.00
MOVJ C00480 BC00480 VJ=20.00
'------------------------
'W29.2
'------------------------
MOVL C00481 BC00481 V=500.0
'------------------------
'W63.5
MACRO1 MJ#(0) ARGF9
'------------------------
SFTOF
SFTON P0301
MOVL C00482 BC00482 V=166.7 PL=0
ARCON
MOVL C00483 BC00483 V=8.3
ARCOF
SFTOF
MOVL C00484 BC00484 V=500.0
MACRO1 MJ#(0) ARGF24
SFTON P0302
MOVL C00485 BC00485 V=166.7 PL=0
ARCON
MOVL C00486 BC00486 V=8.3
ARCOF
MOVL C00487 BC00487 V=166.7 PL=0
SFTOF
MOVL C00488 BC00488 V=500.0
SFTON P0303
MOVL C00489 BC00489 V=166.7 PL=0
ARCON
MOVL C00490 BC00490 V=8.3
ARCOF
SFTOF
MOVL C00491 BC00491 V=166.7 PL=0
MOVL C00492 BC00492 V=500.0
MOVJ C00493 BC00493 VJ=30.00
MOVJ C00494 BC00494 VJ=20.00
MOVJ C00495 BC00495 VJ=30.00
MOVJ C00496 BC00496 VJ=30.00
MOVL C00497 BC00497 V=500.0
'------------------------
'W29.14
'------------------------
SFTON P0304
MOVL C00498 BC00498 V=166.7 PL=0
ARCON
MOVL C00499 BC00499 V=8.3
ARCOF
MOVL C00500 BC00500 V=166.7 PL=0
SFTOF
'PRZEJAZD
MOVL C00501 BC00501 V=500.0
MOVL C00502 BC00502 V=500.0
'------------------------
'W63.17
'------------------------
SFTON P0305
MOVL C00503 BC00503 V=166.7 PL=0
ARCON
MOVL C00504 BC00504 V=8.3
ARCOF
MOVL C00505 BC00505 V=166.7 PL=0
SFTOF
MOVL C00506 BC00506 V=500.0
SFTON P0306
MOVL C00507 BC00507 V=166.7
ARCON
MOVL C00508 BC00508 V=8.3
ARCOF
MOVL C00509 BC00509 V=166.7 PL=0
SFTOF
'PRZEJAZD
MOVL C00510 BC00510 V=500.0
SFTON P0307
MOVL C00511 BC00511 V=166.7
ARCON
MOVL C00512 BC00512 V=8.3
ARCOF
MOVL C00513 BC00513 V=166.7 PL=0
SFTOF
MOVJ C00514 BC00514 VJ=20.00
MOVJ C00515 BC00515 VJ=20.00
MOVJ C00516 BC00516 VJ=30.00
MOVJ C00517 BC00517 VJ=30.00
MOVL C00518 BC00518 V=500.0
'------------------------
'W63.20
'------------------------
SFTON P0308
MOVL C00519 BC00519 V=166.7 PL=0
ARCON
MOVL C00520 BC00520 V=8.3
ARCOF
MOVL C00521 BC00521 V=166.7 PL=0
SFTOF
'PRZEJAZD
MOVL C00522 BC00522 V=500.0
'------------------------
'W63.23
'------------------------
SFTON P0309
MOVL C00523 BC00523 V=166.7 PL=0
ARCON
MOVL C00524 BC00524 V=8.3
ARCOF
MOVL C00525 BC00525 V=250.0 PL=0
SFTOF
MOVL C00526 BC00526 V=500.0
SFTON P0310
MOVL C00527 BC00527 V=166.7 PL=0
ARCON
MOVL C00528 BC00528 V=8.3
ARCOF
MOVL C00529 BC00529 V=250.0 PL=0
SFTOF
MOVL C00530 BC00530 V=500.0
SFTON P0311
MOVL C00531 BC00531 V=166.7 PL=0
ARCON
MOVL C00532 BC00532 V=8.3
ARCOF
MOVL C00533 BC00533 V=250.0 PL=0
SFTOF
MOVL C00534 BC00534 V=500.0
MOVL C00535 BC00535 V=500.0
COMM MOVL C00536 BC00536 V=333.3
COMM '------------------------
COMM 'W29.29
COMM '------------------------
COMM MOVL C00537 BC00537 V=500.0
COMM SFTON P0312
COMM MOVL C00538 BC00538 V=166.7 PL=0
COMM ARCON
COMM MOVL C00539 BC00539 V=8.3
COMM ARCOF
COMM MOVL C00540 BC00540 V=250.0 PL=0
COMM MOVL C00541 BC00541 V=500.0
SFTON P0312
MOVL C00542 BC00542 V=333.3
MOVL C00543 BC00543 V=166.7
ARCON
MOVL C00544 BC00544 V=8.3
ARCOF
SFTOF
'PRZEJAZD
MOVL C00545 BC00545 V=333.3
'PRZEJAZD
'KONIEC SPAWANIA CZESCI WSPOLNEJ
MOVJ C00546 BC00546 VJ=20.00
MOVJ C00547 BC00547 VJ=50.00
MOVJ C00548 BC00548 VJ=20.00
MOVJ C00549 BC00549 VJ=10.00
MOVJ C00550 BC00550 VJ=20.00
MOVJ C00551 BC00551 VJ=20.00
'------------------------
'W28.2
'------------------------
MOVJ C00552 BC00552 VJ=10.00
MOVJ C00553 BC00553 VJ=10.00
MOVL C00554 BC00554 V=500.0
MOVL C00555 BC00555 V=500.0
'------------------------
'W62.5
'------------------------
SFTON P0351
MOVL C00556 BC00556 V=166.7 PL=0
ARCON
MOVL C00557 BC00557 V=8.3
ARCOF
MOVL C00558 BC00558 V=250.0 PL=0
SFTOF
'PRZEJAZD
MOVL C00559 BC00559 V=500.0
MOVL C00560 BC00560 V=500.0
MOVL C00561 BC00561 V=500.0
SFTON P0352
MOVL C00562 BC00562 V=166.7 PL=0
ARCON
MOVL C00563 BC00563 V=8.3
ARCOF
MOVL C00564 BC00564 V=250.0 PL=0
SFTOF
MOVL C00565 BC00565 V=500.0
'------------------------
'W29.8
'------------------------
SFTON P0353
MOVL C00566 BC00566 V=166.7 PL=0
ARCON
MOVL C00567 BC00567 V=8.3
ARCOF
MOVL C00568 BC00568 V=250.0 PL=0
SFTOF
MOVL C00569 BC00569 V=500.0
'PRZEJAZD
MOVL C00570 BC00570 V=500.0
MOVJ C00571 BC00571 VJ=20.00
MOVL C00572 BC00572 V=500.0
MOVL C00573 BC00573 V=500.0
MOVL C00574 BC00574 V=500.0
'------------------------
'W29.11
'------------------------
SFTON P0354
MOVL C00575 BC00575 V=166.7 PL=0
ARCON
MOVL C00576 BC00576 V=8.3
ARCOF
MOVL C00577 BC00577 V=250.0 PL=0
SFTOF
'PRZEJAZD
MOVL C00578 BC00578 V=500.0
'------------------------
'W29.14
'------------------------
SFTON P0355
MOVL C00579 BC00579 V=166.7 PL=0
ARCON
MOVL C00580 BC00580 V=8.3
ARCOF
MOVL C00581 BC00581 V=250.0 PL=0
SFTOF
'PRZEJAZD
MOVL C00582 BC00582 V=500.0
'------------------------
'W63.17
'------------------------
SFTON P0356
MOVL C00583 BC00583 V=166.7 PL=0
ARCON
MOVL C00584 BC00584 V=8.3
ARCOF
MOVL C00585 BC00585 V=250.0 PL=0
SFTOF
MOVL C00586 BC00586 V=500.0
SFTON P0357
MOVL C00587 BC00587 V=166.7 PL=0
ARCON
MOVL C00588 BC00588 V=8.3
ARCOF
MOVL C00589 BC00589 V=250.0 PL=0
SFTOF
'PRZEJAZD
MOVL C00590 BC00590 V=500.0
MOVJ C00591 BC00591 VJ=30.00
MOVJ C00592 BC00592 VJ=30.00
MOVJ C00593 BC00593 VJ=30.00
MOVL C00594 BC00594 V=500.0
MOVL C00595 BC00595 V=500.0
'------------------------
'W62.20
'------------------------
SFTON P0358
MOVL C00596 BC00596 V=166.7 PL=0
ARCON
MOVL C00597 BC00597 V=8.3
ARCOF
MOVL C00598 BC00598 V=250.0 PL=0
SFTOF
'PRZEJAZD
MOVL C00599 BC00599 V=500.0
'------------------------
'W63.23
'------------------------
SFTON P0359
MOVL C00600 BC00600 V=166.7 PL=0
ARCON
MOVL C00601 BC00601 V=8.3
ARCOF
MOVL C00602 BC00602 V=250.0 PL=0
MOVL C00603 BC00603 V=500.0
'------------------------
'W29.29
'------------------------
SFTON P0360
MOVL C00604 BC00604 V=166.7 PL=0
ARCON
MOVL C00605 BC00605 V=8.3
ARCOF
MOVL C00606 BC00606 V=250.0 PL=0
SFTOF
'PRZEJAZD
MOVL C00607 BC00607 V=500.0
SFTON P0361
MOVL C00608 BC00608 V=166.7 PL=0
ARCON
MOVL C00609 BC00609 V=8.3
ARCOF
MOVL C00610 BC00610 V=250.0 PL=0
SFTOF
'------------------------
'W29.32
'------------------------
'PRZEJAZD
MOVL C00611 BC00611 V=500.0
MOVL C00612 BC00612 V=500.0
COMM MOVL C00613 BC00613 V=416.7
COMM MOVL C00614 BC00614 V=500.0
COMM SFTON P0362
COMM MOVL C00615 BC00615 V=166.7 PL=0
COMM ARCON
COMM MOVL C00616 BC00616 V=8.3
COMM ARCOF
COMM MOVL C00617 BC00617 V=250.0 PL=0
COMM MOVL C00618 BC00618 V=500.0
SFTON P0362
MOVL C00619 BC00619 V=333.3
MOVL C00620 BC00620 V=166.7
ARCON
MOVL C00621 BC00621 V=8.3
ARCOF
MOVL C00622 BC00622 V=250.0
SFTOF
MOVJ C00623 BC00623 VJ=20.00
MOVJ C00624 BC00624 VJ=30.00
MOVJ C00625 BC00625 VJ=30.00
MOVJ C00626 BC00626 VJ=30.00
CALL JOB:MOVE_OUT_OF_TUNNEL
END
